LIN {X 0,Y 573.238,Z 498.079,A -85,B 0,C 180,E1 -2309.114,E2 -2309.114} C_VEL
LIN {X 0,Y 573.258,Z 498.071,A -85,B 0,C 180,E1 -2311.967,E2 -2311.967} C_VEL
LIN {X 0,Y 573.252,Z 498.078,A -85,B 0,C 180,E1 -2314.589,E2 -2314.589} C_VEL
LIN {X 0,Y 573.231,Z 498.075,A -85,B 0,C 180,E1 -2317.662,E2 -2317.662} C_VEL
LIN {X 0,Y 573.249,Z 498.072,A -85,B 0,C 180,E1 -2319.923,E2 -2319.923} C_VEL
LIN {X 0,Y 573.254,Z 498.081,A -85,B 0,C 180,E1 -2322.988,E2 -2322.988} C_VEL
LIN {X 0,Y 573.263,Z 498.071,A -85,B 0,C 180,E1 -2325.806,E2 -2325.806} C_VEL
LIN {X 0,Y 573.274,Z 498.076,A -85,B 0,C 180,E1 -2328.734,E2 -2328.734} C_VEL
LIN {X 0,Y 573.299,Z 498.068,A -85,B 0,C 180,E1 -2331.54,E2 -2331.54} C_VEL
LIN {X 0,Y 573.291,Z 498.068,A -85,B 0,C 180,E1 -2334.371,E2 -2334.371} C_VEL
LIN {X 0,Y 573.3,Z 498.066,A -85,B 0,C 180,E1 -2337.892,E2 -2337.892} C_VEL
LIN {X 0,Y 573.329,Z 498.067,A -85,B 0,C 180,E1 -2340.702,E2 -2340.702} C_VEL
LIN {X 0,Y 573.239,Z 498.077,A -85,B 0,C 180,E1 -2343.514,E2 -2343.514} C_VEL
LIN {X 0,Y 573.294,Z 498.069,A -85,B 0,C 180,E1 -2345.628,E2 -2345.628} C_VEL
LIN {X 0,Y 573.299,Z 498.068,A -85,B 0,C 180,E1 -2348.459,E2 -2348.459} C_VEL
LIN {X 0,Y 573.288,Z 498.074,A -85,B 0,C 180,E1 -2351.311,E2 -2351.311} C_VEL
LIN {X 0,Y 573.27,Z 498.071,A -85,B 0,C 180,E1 -2354.425,E2 -2354.425} C_VEL
LIN {X 0,Y 573.25,Z 498.083,A -85,B 0,C 180,E1 -2357.111,E2 -2357.111} C_VEL
LIN {X 0,Y 573.248,Z 498.073,A -85,B 0,C 180,E1 -2360.076,E2 -2360.076} C_VEL
LIN {X 0,Y 573.23,Z 498.076,A -85,B 0,C 180,E1 -2362.338,E2 -2362.338} C_VEL
LIN {X 0,Y 573.242,Z 498.075,A -85,B 0,C 180,E1 -2364.401,E2 -2364.401} C_VEL
LIN {X 0,Y 572.616,Z 498.16,A -85,B 0,C 180,E1 -2364.988,E2 -2364.988} C_VEL
LIN {X 0,Y 569.779,Z 498.518,A -85,B 0,C 180,E1 -2365.939,E2 -2365.939} C_VEL
LIN {X 0,Y 567.351,Z 498.821,A -85,B 0,C 180,E1 -2366.705,E2 -2366.705} C_VEL
LIN {X 0,Y 566.298,Z 498.949,A -85,B 0,C 180,E1 -2367.297,E2 -2367.297} C_VEL
LIN {X 0,Y 566.208,Z 498.956,A -85,B 0,C 180,E1 -2367.497,E2 -2367.497} C_VEL
LIN {X 0,Y 566.186,Z 498.955,A -85,B 0,C 180,E1 -2370.592,E2 -2370.592} C_VEL
LIN {X 0,Y 566.22,Z 498.958,A -85,B 0,C 180,E1 -2373.102,E2 -2373.102} C_VEL
LIN {X 0,Y 566.261,Z 499.123,A -85,B 0,C 180,E1 -2374.382,E2 -2374.382} C_VEL
LIN {X 0,Y 566.267,Z 510.219,A -85,B 0,C 180,E1 -2376.564,E2 -2376.564} C_VEL
LIN {X 0,Y 566.196,Z 517.853,A -85,B 0,C 180,E1 -2378.051,E2 -2378.051} C_VEL
LIN {X 0,Y 567.197,Z 524.442,A -85,B 0,C 180,E1 -2378.169,E2 -2378.169} C_VEL
LIN {X 0,Y 566.927,Z 624.641,A -85,B 0,C 180,E1 -2379.461,E2 -2379.461} C_VEL
LIN {X 0,Y 566.843,Z 638.116,A -85,B 0,C 180,E1 -2379.791,E2 -2379.791} C_VEL
LIN {X 0,Y 566.739,Z 649.818,A -85,B 0,C 180,E1 -2380.211,E2 -2380.211} C_VEL
LIN {X 0,Y 566.583,Z 661.36,A -85,B 0,C 180,E1 -2380.764,E2 -2380.764} C_VEL
LIN {X 0,Y 566.456,Z 672.754,A -85,B 0,C 180,E1 -2381.469,E2 -2381.469} C_VEL
LIN {X 0,Y 566.307,Z 683.695,A -85,B 0,C 180,E1 -2382.318,E2 -2382.318} C_VEL
LIN {X 0,Y 566.189,Z 693.549,A -85,B 0,C 180,E1 -2383.273,E2 -2383.273} C_VEL
LIN {X 0,Y 566.069,Z 701.912,A -85,B 0,C 180,E1 -2384.272,E2 -2384.272} C_VEL
LIN {X 0,Y 566.024,Z 708.75,A -85,B 0,C 180,E1 -2385.273,E2 -2385.273} C_VEL
LIN {X 0,Y 565.94,Z 715.445,A -85,B 0,C 180,E1 -2386.498,E2 -2386.498} C_VEL
LIN {X 0,Y 565.918,Z 719.703,A -85,B 0,C 180,E1 -2387.498,E2 -2387.498} C_VEL
LIN {X 0,Y 565.921,Z 722.017,A -85,B 0,C 180,E1 -2388.169,E2 -2388.169} C_VEL
LIN {X 0,Y 565.836,Z 724.94,A -85,B 0,C 180,E1 -2389.257,E2 -2389.257} C_VEL
LIN {X 0,Y 565.848,Z 726.888,A -85,B 0,C 180,E1 -2390.358,E2 -2390.358} C_VEL
LIN {X 0,Y 565.827,Z 727.91,A -85,B 0,C 180,E1 -2391.609,E2 -2391.609} C_VEL
LIN {X 0,Y 565.828,Z 727.856,A -85,B 0,C 180,E1 -2392.648,E2 -2392.648} C_VEL
LIN {X 0,Y 565.816,Z 726.731,A -85,B 0,C 180,E1 -2393.839,E2 -2393.839} C_VEL
LIN {X 0,Y 565.872,Z 724.149,A -85,B 0,C 180,E1 -2395.159,E2 -2395.159} C_VEL
LIN {X 0,Y 565.916,Z 720.706,A -85,B 0,C 180,E1 -2396.31,E2 -2396.31} C_VEL
LIN {X 0,Y 565.946,Z 715.36,A -85,B 0,C 180,E1 -2397.61,E2 -2397.61} C_VEL
LIN {X 0,Y 565.995,Z 708.949,A -85,B 0,C 180,E1 -2398.786,E2 -2398.786} C_VEL
LIN {X 0,Y 566.094,Z 701.93,A -85,B 0,C 180,E1 -2399.815,E2 -2399.815} C_VEL
LIN {X 0,Y 566.175,Z 693.319,A -85,B 0,C 180,E1 -2400.843,E2 -2400.843} C_VEL
LIN {X 0,Y 566.319,Z 683.652,A -85,B 0,C 180,E1 -2401.775,E2 -2401.775} C_VEL
LIN {X 0,Y 566.432,Z 673.445,A -85,B 0,C 180,E1 -2402.573,E2 -2402.573} C_VEL
LIN {X 0,Y 566.569,Z 662.396,A -85,B 0,C 180,E1 -2403.267,E2 -2403.267} C_VEL
LIN {X 0,Y 566.717,Z 650.965,A -85,B 0,C 180,E1 -2403.832,E2 -2403.832} C_VEL
LIN {X 0,Y 566.828,Z 638.084,A -85,B 0,C 180,E1 -2404.301,E2 -2404.301} C_VEL
LIN {X 0,Y 566.939,Z 625.415,A -85,B 0,C 180,E1 -2404.613,E2 -2404.613} C_VEL
LIN {X 0,Y 567.029,Z 594.146,A -85,B 0,C 180,E1 -2405.036,E2 -2405.036} C_VEL
LIN {X 0,Y 567.13,Z 523.477,A -85,B 0,C 180,E1 -2405.935,E2 -2405.935} C_VEL
LIN {X 0,Y 566.222,Z 517.846,A -85,B 0,C 180,E1 -2406.04,E2 -2406.04} C_VEL
LIN {X 0,Y 566.357,Z 503.159,A -85,B 0,C 180,E1 -2408.909,E2 -2408.909} C_VEL
LIN {X 0,Y 566.225,Z 498.953,A -85,B 0,C 180,E1 -2409.759,E2 -2409.759} C_VEL
LIN {X 0,Y 566.222,Z 498.958,A -85,B 0,C 180,E1 -2412.886,E2 -2412.886} C_VEL
LIN {X 0,Y 566.231,Z 498.947,A -85,B 0,C 180,E1 -2415.627,E2 -2415.627} C_VEL
LIN {X 0,Y 566.232,Z 498.953,A -85,B 0,C 180,E1 -2418.675,E2 -2418.675} C_VEL
LIN {X 0,Y 566.226,Z 498.95,A -85,B 0,C 180,E1 -2421.434,E2 -2421.434} C_VEL
LIN {X 0,Y 566.263,Z 498.944,A -85,B 0,C 180,E1 -2424.302,E2 -2424.302} C_VEL
LIN {X 0,Y 566.282,Z 498.94,A -85,B 0,C 180,E1 -2427.866,E2 -2427.866} C_VEL
LIN {X 0,Y 566.302,Z 498.945,A -85,B 0,C 180,E1 -2430.711,E2 -2430.711} C_VEL
LIN {X 0,Y 566.271,Z 498.951,A -85,B 0,C 180,E1 -2432.845,E2 -2432.845} C_VEL
LIN {X 0,Y 566.264,Z 498.943,A -85,B 0,C 180,E1 -2435.698,E2 -2435.698} C_VEL
LIN {X 0,Y 566.231,Z 498.951,A -85,B 0,C 180,E1 -2438.565,E2 -2438.565} C_VEL
LIN {X 0,Y 566.239,Z 498.948,A -85,B 0,C 180,E1 -2441.454,E2 -2441.454} C_VEL
LIN {X 0,Y 566.231,Z 498.95,A -85,B 0,C 180,E1 -2444.507,E2 -2444.507} C_VEL
LIN {X 0,Y 566.2,Z 498.955,A -85,B 0,C 180,E1 -2447.331,E2 -2447.331} C_VEL
LIN {X 0,Y 566.211,Z 498.951,A -85,B 0,C 180,E1 -2450.337,E2 -2450.337} C_VEL
LIN {X 0,Y 566.185,Z 498.956,A -85,B 0,C 180,E1 -2453.403,E2 -2453.403} C_VEL
LIN {X 0,Y 566.21,Z 498.95,A -85,B 0,C 180,E1 -2455.749,E2 -2455.749} C_VEL
LIN {X 0,Y 566.201,Z 498.951,A -85,B 0,C 180,E1 -2458.203,E2 -2458.203} C_VEL
LIN {X 0,Y 566.19,Z 498.955,A -85,B 0,C 180,E1 -2460.591,E2 -2460.591} C_VEL
LIN {X 0,Y 566.223,Z 498.957,A -85,B 0,C 180,E1 -2463.101,E2 -2463.101} C_VEL
LIN {X 0,Y 566.206,Z 498.951,A -85,B 0,C 180,E1 -2465.688,E2 -2465.688} C_VEL
LIN {X 0,Y 566.211,Z 498.952,A -85,B 0,C 180,E1 -2468.559,E2 -2468.559} C_VEL
LIN {X 0,Y 566.214,Z 498.958,A -85,B 0,C 180,E1 -2471.135,E2 -2471.135} C_VEL
LIN {X 0,Y 566.193,Z 498.951,A -85,B 0,C 180,E1 -2474.035,E2 -2474.035} C_VEL
LIN {X 0,Y 566.197,Z 498.961,A -85,B 0,C 180,E1 -2477.082,E2 -2477.082} C_VEL
LIN {X 0,Y 566.219,Z 498.949,A -85,B 0,C 180,E1 -2479.802,E2 -2479.802} C_VEL
LIN {X 0,Y 566.19,Z 498.955,A -85,B 0,C 180,E1 -2482.599,E2 -2482.599} C_VEL
LIN {X 0,Y 566.215,Z 498.958,A -85,B 0,C 180,E1 -2485.183,E2 -2485.183} C_VEL
LIN {X 0,Y 566.226,Z 498.949,A -85,B 0,C 180,E1 -2487.744,E2 -2487.744} C_VEL
LIN {X 0,Y 566.22,Z 498.949,A -85,B 0,C 180,E1 -2490.323,E2 -2490.323} C_VEL
LIN {X 0,Y 566.228,Z 498.954,A -85,B 0,C 180,E1 -2493.334,E2 -2493.334} C_VEL
LIN {X 0,Y 566.19,Z 498.953,A -85,B 0,C 180,E1 -2495.819,E2 -2495.819} C_VEL
LIN {X 0,Y 566.207,Z 498.956,A -85,B 0,C 180,E1 -2498.903,E2 -2498.903} C_VEL
LIN {X 0,Y 566.205,Z 498.96,A -85,B 0,C 180,E1 -2501.173,E2 -2501.173} C_VEL
LIN {X 0,Y 566.212,Z 498.955,A -85,B 0,C 180,E1 -2503.413,E2 -2503.413} C_VEL
LIN {X 0,Y 566.192,Z 498.952,A -85,B 0,C 180,E1 -2506.359,E2 -2506.359} C_VEL
LIN {X 0,Y 566.264,Z 498.945,A -85,B 0,C 180,E1 -2508.654,E2 -2508.654} C_VEL
LIN {X 0,Y 566.241,Z 498.951,A -85,B 0,C 180,E1 -2511.435,E2 -2511.435} C_VEL
LIN {X 0,Y 566.259,Z 498.943,A -85,B 0,C 180,E1 -2514.302,E2 -2514.302} C_VEL
LIN {X 0,Y 566.271,Z 498.943,A -85,B 0,C 180,E1 -2517.867,E2 -2517.867} C_VEL
LIN {X 0,Y 566.3,Z 498.941,A -85,B 0,C 180,E1 -2520.711,E2 -2520.711} C_VEL
LIN {X 0,Y 566.274,Z 498.946,A -85,B 0,C 180,E1 -2522.846,E2 -2522.846} C_VEL
LIN {X 0,Y 566.263,Z 498.946,A -85,B 0,C 180,E1 -2525.699,E2 -2525.699} C_VEL
LIN {X 0,Y 566.242,Z 498.946,A -85,B 0,C 180,E1 -2528.566,E2 -2528.566} C_VEL
LIN {X 0,Y 566.242,Z 498.952,A -85,B 0,C 180,E1 -2531.455,E2 -2531.455} C_VEL
LIN {X 0,Y 566.225,Z 498.948,A -85,B 0,C 180,E1 -2534.508,E2 -2534.508} C_VEL
LIN {X 0,Y 566.198,Z 498.96,A -85,B 0,C 180,E1 -2537.332,E2 -2537.332} C_VEL
LIN {X 0,Y 566.212,Z 498.949,A -85,B 0,C 180,E1 -2540.338,E2 -2540.338} C_VEL
LIN {X 0,Y 566.182,Z 498.961,A -85,B 0,C 180,E1 -2543.405,E2 -2543.405} C_VEL
LIN {X 0,Y 566.219,Z 498.951,A -85,B 0,C 180,E1 -2545.749,E2 -2545.749} C_VEL
LIN {X 0,Y 566.2,Z 498.951,A -85,B 0,C 180,E1 -2548.204,E2 -2548.204} C_VEL
LIN {X 0,Y 566.188,Z 498.953,A -85,B 0,C 180,E1 -2550.593,E2 -2550.593} C_VEL
LIN {X 0,Y 566.223,Z 498.954,A -85,B 0,C 180,E1 -2553.102,E2 -2553.102} C_VEL
LIN {X 0,Y 566.208,Z 498.954,A -85,B 0,C 180,E1 -2555.689,E2 -2555.689} C_VEL
LIN {X 0,Y 566.212,Z 498.95,A -85,B 0,C 180,E1 -2558.56,E2 -2558.56} C_VEL
LIN {X 0,Y 566.208,Z 498.956,A -85,B 0,C 180,E1 -2561.137,E2 -2561.137} C_VEL
LIN {X 0,Y 566.196,Z 498.952,A -85,B 0,C 180,E1 -2564.036,E2 -2564.036} C_VEL
LIN {X 0,Y 566.207,Z 498.955,A -85,B 0,C 180,E1 -2567.083,E2 -2567.083} C_VEL
LIN {X 0,Y 566.225,Z 498.951,A -85,B 0,C 180,E1 -2569.804,E2 -2569.804} C_VEL
LIN {X 0,Y 566.198,Z 498.951,A -85,B 0,C 180,E1 -2572.6,E2 -2572.6} C_VEL
LIN {X 0,Y 566.209,Z 498.956,A -85,B 0,C 180,E1 -2575.183,E2 -2575.183} C_VEL
LIN {X 0,Y 566.234,Z 498.952,A -85,B 0,C 180,E1 -2577.745,E2 -2577.745} C_VEL
LIN {X 0,Y 566.204,Z 498.951,A -85,B 0,C 180,E1 -2580.329,E2 -2580.329} C_VEL
LIN {X 0,Y 566.212,Z 498.952,A -85,B 0,C 180,E1 -2582.662,E2 -2582.662} C_VEL
LIN {X 0,Y 566.249,Z 499.022,A -85,B 0,C 180,E1 -2585.456,E2 -2585.456} C_VEL
LIN {X 0,Y 567.269,Z 504.225,A -85,B 0,C 180,E1 -2586.221,E2 -2586.221} C_VEL
LIN {X 0,Y 567.127,Z 520.193,A -85,B 0,C 180,E1 -2588.465,E2 -2588.465} C_VEL
LIN {X 0,Y 566.837,Z 539.96,A -85,B 0,C 180,E1 -2591.195,E2 -2591.195} C_VEL
LIN {X 0,Y 566.582,Z 560.431,A -85,B 0,C 180,E1 -2593.979,E2 -2593.979} C_VEL
LIN {X 0,Y 566.428,Z 575.357,A -85,B 0,C 180,E1 -2595.987,E2 -2595.987} C_VEL
LIN {X 0,Y 567.197,Z 581.535,A -85,B 0,C 180,E1 -2596.087,E2 -2596.087} C_VEL
LIN {X 0,Y 566.921,Z 683.962,A -85,B 0,C 180,E1 -2597.403,E2 -2597.403} C_VEL
LIN {X 0,Y 566.848,Z 697.229,A -85,B 0,C 180,E1 -2597.719,E2 -2597.719} C_VEL
LIN {X 0,Y 566.758,Z 709.382,A -85,B 0,C 180,E1 -2598.149,E2 -2598.149} C_VEL
LIN {X 0,Y 566.627,Z 721.158,A -85,B 0,C 180,E1 -2598.708,E2 -2598.708} C_VEL
LIN {X 0,Y 566.458,Z 733.205,A -85,B 0,C 180,E1 -2599.456,E2 -2599.456} C_VEL
LIN {X 0,Y 566.318,Z 743.604,A -85,B 0,C 180,E1 -2600.266,E2 -2600.266} C_VEL
LIN {X 0,Y 566.207,Z 752.115,A -85,B 0,C 180,E1 -2601.074,E2 -2601.074} C_VEL
LIN {X 0,Y 566.112,Z 759.962,A -85,B 0,C 180,E1 -2601.972,E2 -2601.972} C_VEL
LIN {X 0,Y 566.004,Z 767.623,A -85,B 0,C 180,E1 -2603.047,E2 -2603.047} C_VEL
LIN {X 0,Y 566.004,Z 774.681,A -85,B 0,C 180,E1 -2604.299,E2 -2604.299} C_VEL
LIN {X 0,Y 565.933,Z 779.372,A -85,B 0,C 180,E1 -2605.37,E2 -2605.37} C_VEL
LIN {X 0,Y 565.927,Z 782.958,A -85,B 0,C 180,E1 -2606.44,E2 -2606.44} C_VEL
LIN {X 0,Y 565.878,Z 784.808,A -85,B 0,C 180,E1 -2607.153,E2 -2607.153} C_VEL
LIN {X 0,Y 565.846,Z 787.186,A -85,B 0,C 180,E1 -2608.577,E2 -2608.577} C_VEL
LIN {X 0,Y 565.839,Z 788,A -85,B 0,C 180,E1 -2610,E2 -2610} C_VEL
LIN {X 0,Y 565.846,Z 787.186,A -85,B 0,C 180,E1 -2611.423,E2 -2611.423} C_VEL
LIN {X 0,Y 565.878,Z 784.81,A -85,B 0,C 180,E1 -2612.847,E2 -2612.847} C_VEL
LIN {X 0,Y 565.926,Z 781.896,A -85,B 0,C 180,E1 -2613.916,E2 -2613.916} C_VEL
LIN {X 0,Y 565.878,Z 777.949,A -85,B 0,C 180,E1 -2614.987,E2 -2614.987} C_VEL
LIN {X 0,Y 566.002,Z 772.867,A -85,B 0,C 180,E1 -2616.058,E2 -2616.058} C_VEL
LIN {X 0,Y 566.04,Z 766.47,A -85,B 0,C 180,E1 -2617.132,E2 -2617.132} C_VEL
LIN {X 0,Y 566.134,Z 758.48,A -85,B 0,C 180,E1 -2618.207,E2 -2618.207} C_VEL
LIN {X 0,Y 566.228,Z 750.338,A -85,B 0,C 180,E1 -2619.105,E2 -2619.105} C_VEL
LIN {X 0,Y 566.341,Z 740.404,A -85,B 0,C 180,E1 -2620.005,E2 -2620.005} C_VEL
LIN {X 0,Y 566.523,Z 729.288,A -85,B 0,C 180,E1 -2620.807,E2 -2620.807} C_VEL
LIN {X 0,Y 566.66,Z 718.182,A -85,B 0,C 180,E1 -2621.445,E2 -2621.445} C_VEL
LIN {X 0,Y 566.735,Z 705.991,A -85,B 0,C 180,E1 -2621.988,E2 -2621.988} C_VEL
LIN {X 0,Y 566.879,Z 693.188,A -85,B 0,C 180,E1 -2622.394,E2 -2622.394} C_VEL
LIN {X 0,Y 566.988,Z 681.127,A -85,B 0,C 180,E1 -2622.641,E2 -2622.641} C_VEL
LIN {X 0,Y 567.056,Z 579.746,A -85,B 0,C 180,E1 -2623.94,E2 -2623.94} C_VEL
LIN {X 0,Y 566.446,Z 575.272,A -85,B 0,C 180,E1 -2624.024,E2 -2624.024} C_VEL
LIN {X 0,Y 566.673,Z 552.206,A -85,B 0,C 180,E1 -2627.135,E2 -2627.135} C_VEL
LIN {X 0,Y 566.955,Z 530.408,A -85,B 0,C 180,E1 -2630.119,E2 -2630.119} C_VEL
LIN {X 0,Y 567.305,Z 509.936,A -85,B 0,C 180,E1 -2632.969,E2 -2632.969} C_VEL
LIN {X 0,Y 567.276,Z 504.204,A -85,B 0,C 180,E1 -2633.782,E2 -2633.782} C_VEL
LIN {X 0,Y 566.257,Z 498.954,A -85,B 0,C 180,E1 -2634.568,E2 -2634.568} C_VEL
LIN {X 0,Y 566.212,Z 498.952,A -85,B 0,C 180,E1 -2637.338,E2 -2637.338} C_VEL
LIN {X 0,Y 566.202,Z 498.952,A -85,B 0,C 180,E1 -2639.768,E2 -2639.768} C_VEL
LIN {X 0,Y 566.207,Z 498.958,A -85,B 0,C 180,E1 -2642.43,E2 -2642.43} C_VEL
LIN {X 0,Y 566.212,Z 498.955,A -85,B 0,C 180,E1 -2644.994,E2 -2644.994} C_VEL
LIN {X 0,Y 566.196,Z 498.952,A -85,B 0,C 180,E1 -2647.46,E2 -2647.46} C_VEL
LIN {X 0,Y 566.225,Z 498.951,A -85,B 0,C 180,E1 -2650.196,E2 -2650.196} C_VEL
LIN {X 0,Y 566.207,Z 498.955,A -85,B 0,C 180,E1 -2653.052,E2 -2653.052} C_VEL
LIN {X 0,Y 566.198,Z 498.952,A -85,B 0,C 180,E1 -2656.047,E2 -2656.047} C_VEL
LIN {X 0,Y 566.207,Z 498.958,A -85,B 0,C 180,E1 -2658.863,E2 -2658.863} C_VEL
LIN {X 0,Y 566.186,Z 498.953,A -85,B 0,C 180,E1 -2661.636,E2 -2661.636} C_VEL
LIN {X 0,Y 566.208,Z 498.953,A -85,B 0,C 180,E1 -2664.311,E2 -2664.311} C_VEL
LIN {X 0,Y 566.223,Z 498.957,A -85,B 0,C 180,E1 -2666.898,E2 -2666.898} C_VEL
LIN {X 0,Y 566.188,Z 498.954,A -85,B 0,C 180,E1 -2669.407,E2 -2669.407} C_VEL
LIN {X 0,Y 566.221,Z 498.948,A -85,B 0,C 180,E1 -2671.858,E2 -2671.858} C_VEL
LIN {X 0,Y 566.22,Z 498.95,A -85,B 0,C 180,E1 -2674.251,E2 -2674.251} C_VEL
LIN {X 0,Y 566.185,Z 498.959,A -85,B 0,C 180,E1 -2676.713,E2 -2676.713} C_VEL
LIN {X 0,Y 566.212,Z 498.949,A -85,B 0,C 180,E1 -2679.662,E2 -2679.662} C_VEL
LIN {X 0,Y 566.196,Z 498.957,A -85,B 0,C 180,E1 -2682.668,E2 -2682.668} C_VEL
LIN {X 0,Y 566.224,Z 498.948,A -85,B 0,C 180,E1 -2685.626,E2 -2685.626} C_VEL
LIN {X 0,Y 566.266,Z 498.948,A -85,B 0,C 180,E1 -2688.653,E2 -2688.653} C_VEL
LIN {X 0,Y 566.24,Z 498.949,A -85,B 0,C 180,E1 -2691.434,E2 -2691.434} C_VEL
LIN {X 0,Y 566.259,Z 498.944,A -85,B 0,C 180,E1 -2694.301,E2 -2694.301} C_VEL
LIN {X 0,Y 566.271,Z 498.942,A -85,B 0,C 180,E1 -2697.866,E2 -2697.866} C_VEL
LIN {X 0,Y 566.299,Z 498.943,A -85,B 0,C 180,E1 -2700.711,E2 -2700.711} C_VEL
LIN {X 0,Y 566.272,Z 498.949,A -85,B 0,C 180,E1 -2702.845,E2 -2702.845} C_VEL
LIN {X 0,Y 566.262,Z 498.944,A -85,B 0,C 180,E1 -2705.698,E2 -2705.698} C_VEL
LIN {X 0,Y 566.241,Z 498.948,A -85,B 0,C 180,E1 -2708.565,E2 -2708.565} C_VEL
LIN {X 0,Y 566.24,Z 498.95,A -85,B 0,C 180,E1 -2711.454,E2 -2711.454} C_VEL
LIN {X 0,Y 566.223,Z 498.95,A -85,B 0,C 180,E1 -2714.507,E2 -2714.507} C_VEL
LIN {X 0,Y 566.195,Z 498.959,A -85,B 0,C 180,E1 -2717.331,E2 -2717.331} C_VEL
LIN {X 0,Y 566.211,Z 498.95,A -85,B 0,C 180,E1 -2720.337,E2 -2720.337} C_VEL
LIN {X 0,Y 566.18,Z 498.961,A -85,B 0,C 180,E1 -2723.404,E2 -2723.404} C_VEL
LIN {X 0,Y 566.218,Z 498.952,A -85,B 0,C 180,E1 -2725.748,E2 -2725.748} C_VEL
LIN {X 0,Y 566.208,Z 498.956,A -85,B 0,C 180,E1 -2727.497,E2 -2727.497} C_VEL
LIN {X 0,Y 565.529,Z 499.038,A -85,B 0,C 180,E1 -2728.091,E2 -2728.091} C_VEL
LIN {X 0,Y 562.664,Z 499.401,A -85,B 0,C 180,E1 -2729.054,E2 -2729.054} C_VEL
LIN {X 0,Y 560.253,Z 499.696,A -85,B 0,C 180,E1 -2729.83,E2 -2729.83} C_VEL
LIN {X 0,Y 559.225,Z 499.822,A -85,B 0,C 180,E1 -2730.429,E2 -2730.429} C_VEL
LIN {X 0,Y 559.144,Z 499.833,A -85,B 0,C 180,E1 -2730.631,E2 -2730.631} C_VEL
LIN {X 0,Y 559.168,Z 499.835,A -85,B 0,C 180,E1 -2733.574,E2 -2733.574} C_VEL
LIN {X 0,Y 559.223,Z 499.985,A -85,B 0,C 180,E1 -2734.325,E2 -2734.325} C_VEL
LIN {X 0,Y 559.247,Z 510.703,A -85,B 0,C 180,E1 -2736.461,E2 -2736.461} C_VEL
LIN {X 0,Y 559.188,Z 517.827,A -85,B 0,C 180,E1 -2737.867,E2 -2737.867} C_VEL
LIN {X 0,Y 560.336,Z 525.282,A -85,B 0,C 180,E1 -2738.006,E2 -2738.006} C_VEL
LIN {X 0,Y 560.038,Z 624.109,A -85,B 0,C 180,E1 -2739.293,E2 -2739.293} C_VEL
LIN {X 0,Y 559.894,Z 637.137,A -85,B 0,C 180,E1 -2739.607,E2 -2739.607} C_VEL
LIN {X 0,Y 559.783,Z 650.179,A -85,B 0,C 180,E1 -2740.077,E2 -2740.077} C_VEL
LIN {X 0,Y 559.589,Z 662.251,A -85,B 0,C 180,E1 -2740.672,E2 -2740.672} C_VEL
LIN {X 0,Y 559.443,Z 673.522,A -85,B 0,C 180,E1 -2741.389,E2 -2741.389} C_VEL
LIN {X 0,Y 559.273,Z 684.342,A -85,B 0,C 180,E1 -2742.251,E2 -2742.251} C_VEL
LIN {X 0,Y 559.137,Z 693.869,A -85,B 0,C 180,E1 -2743.197,E2 -2743.197} C_VEL
LIN {X 0,Y 559.006,Z 702.977,A -85,B 0,C 180,E1 -2744.316,E2 -2744.316} C_VEL
LIN {X 0,Y 558.94,Z 709.091,A -85,B 0,C 180,E1 -2745.242,E2 -2745.242} C_VEL
LIN {X 0,Y 558.874,Z 714.53,A -85,B 0,C 180,E1 -2746.241,E2 -2746.241} C_VEL
LIN {X 0,Y 558.839,Z 718.865,A -85,B 0,C 180,E1 -2747.227,E2 -2747.227} C_VEL
LIN {X 0,Y 558.819,Z 722.252,A -85,B 0,C 180,E1 -2748.199,E2 -2748.199} C_VEL
LIN {X 0,Y 558.756,Z 724.792,A -85,B 0,C 180,E1 -2749.153,E2 -2749.153} C_VEL
LIN {X 0,Y 558.756,Z 726.547,A -85,B 0,C 180,E1 -2750.107,E2 -2750.107} C_VEL
LIN {X 0,Y 558.725,Z 727.737,A -85,B 0,C 180,E1 -2751.248,E2 -2751.248} C_VEL
LIN {X 0,Y 558.735,Z 727.926,A -85,B 0,C 180,E1 -2752.413,E2 -2752.413} C_VEL
LIN {X 0,Y 558.719,Z 726.879,A -85,B 0,C 180,E1 -2753.759,E2 -2753.759} C_VEL
LIN {X 0,Y 558.762,Z 724.994,A -85,B 0,C 180,E1 -2754.84,E2 -2754.84} C_VEL
LIN {X 0,Y 558.813,Z 721.597,A -85,B 0,C 180,E1 -2756.104,E2 -2756.104} C_VEL
LIN {X 0,Y 558.856,Z 716.567,A -85,B 0,C 180,E1 -2757.412,E2 -2757.412} C_VEL
LIN {X 0,Y 558.919,Z 711.258,A -85,B 0,C 180,E1 -2758.473,E2 -2758.473} C_VEL
LIN {X 0,Y 558.989,Z 704.215,A -85,B 0,C 180,E1 -2759.6,E2 -2759.6} C_VEL
LIN {X 0,Y 559.109,Z 696.087,A -85,B 0,C 180,E1 -2760.645,E2 -2760.645} C_VEL
LIN {X 0,Y 559.234,Z 686.864,A -85,B 0,C 180,E1 -2761.606,E2 -2761.606} C_VEL
LIN {X 0,Y 559.42,Z 676.213,A -85,B 0,C 180,E1 -2762.505,E2 -2762.505} C_VEL
LIN {X 0,Y 559.556,Z 665.137,A -85,B 0,C 180,E1 -2763.25,E2 -2763.25} C_VEL
LIN {X 0,Y 559.712,Z 653.158,A -85,B 0,C 180,E1 -2763.88,E2 -2763.88} C_VEL
LIN {X 0,Y 559.893,Z 640.397,A -85,B 0,C 180,E1 -2764.383,E2 -2764.383} C_VEL
LIN {X 0,Y 560.011,Z 628.043,A -85,B 0,C 180,E1 -2764.718,E2 -2764.718} C_VEL
LIN {X 0,Y 560.089,Z 611.02,A -85,B 0,C 180,E1 -2764.982,E2 -2764.982} C_VEL
LIN {X 0,Y 560.287,Z 524.896,A -85,B 0,C 180,E1 -2766.09,E2 -2766.09} C_VEL
LIN {X 0,Y 559.177,Z 517.889,A -85,B 0,C 180,E1 -2766.212,E2 -2766.212} C_VEL
LIN {X 0,Y 559.324,Z 503.713,A -85,B 0,C 180,E1 -2769.017,E2 -2769.017} C_VEL
LIN {X 0,Y 559.201,Z 499.829,A -85,B 0,C 180,E1 -2769.829,E2 -2769.829} C_VEL
LIN {X 0,Y 559.179,Z 499.831,A -85,B 0,C 180,E1 -2773.198,E2 -2773.198} C_VEL
LIN {X 0,Y 559.171,Z 499.827,A -85,B 0,C 180,E1 -2776.184,E2 -2776.184} C_VEL
LIN {X 0,Y 559.192,Z 499.83,A -85,B 0,C 180,E1 -2779.134,E2 -2779.134} C_VEL
LIN {X 0,Y 559.204,Z 499.822,A -85,B 0,C 180,E1 -2782.054,E2 -2782.054} C_VEL
LIN {X 0,Y 559.252,Z 499.826,A -85,B 0,C 180,E1 -2784.953,E2 -2784.953} C_VEL
LIN {X 0,Y 559.253,Z 499.816,A -85,B 0,C 180,E1 -2787.839,E2 -2787.839} C_VEL
LIN {X 0,Y 559.272,Z 499.82,A -85,B 0,C 180,E1 -2790.72,E2 -2790.72} C_VEL
LIN {X 0,Y 559.237,Z 499.828,A -85,B 0,C 180,E1 -2792.881,E2 -2792.881} C_VEL
LIN {X 0,Y 559.234,Z 499.819,A -85,B 0,C 180,E1 -2795.77,E2 -2795.77} C_VEL
LIN {X 0,Y 559.189,Z 499.83,A -85,B 0,C 180,E1 -2798.674,E2 -2798.674} C_VEL
LIN {X 0,Y 559.203,Z 499.824,A -85,B 0,C 180,E1 -2801.6,E2 -2801.6} C_VEL
LIN {X 0,Y 559.197,Z 499.827,A -85,B 0,C 180,E1 -2804.595,E2 -2804.595} C_VEL
LIN {X 0,Y 559.16,Z 499.829,A -85,B 0,C 180,E1 -2807.556,E2 -2807.556} C_VEL
LIN {X 0,Y 559.169,Z 499.827,A -85,B 0,C 180,E1 -2809.837,E2 -2809.837} C_VEL
LIN {X 0,Y 559.138,Z 499.831,A -85,B 0,C 180,E1 -2812.152,E2 -2812.152} C_VEL
LIN {X 0,Y 559.174,Z 499.833,A -85,B 0,C 180,E1 -2815.187,E2 -2815.187} C_VEL
LIN {X 0,Y 559.188,Z 499.825,A -85,B 0,C 180,E1 -2817.711,E2 -2817.711} C_VEL
LIN {X 0,Y 559.164,Z 499.827,A -85,B 0,C 180,E1 -2820.181,E2 -2820.181} C_VEL
LIN {X 0,Y 559.17,Z 499.831,A -85,B 0,C 180,E1 -2822.713,E2 -2822.713} C_VEL
LIN {X 0,Y 559.151,Z 499.834,A -85,B 0,C 180,E1 -2825.321,E2 -2825.321} C_VEL
LIN {X 0,Y 559.13,Z 499.831,A -85,B 0,C 180,E1 -2828.017,E2 -2828.017} C_VEL
LIN {X 0,Y 559.173,Z 499.832,A -85,B 0,C 180,E1 -2830.81,E2 -2830.81} C_VEL
LIN {X 0,Y 559.157,Z 499.829,A -85,B 0,C 180,E1 -2833.731,E2 -2833.731} C_VEL
LIN {X 0,Y 559.16,Z 499.833,A -85,B 0,C 180,E1 -2836.801,E2 -2836.801} C_VEL
LIN {X 0,Y 559.168,Z 499.835,A -85,B 0,C 180,E1 -2839.189,E2 -2839.189} C_VEL
LIN {X 0,Y 559.127,Z 499.832,A -85,B 0,C 180,E1 -2841.982,E2 -2841.982} C_VEL
LIN {X 0,Y 559.151,Z 499.832,A -85,B 0,C 180,E1 -2844.678,E2 -2844.678} C_VEL
LIN {X 0,Y 559.165,Z 499.833,A -85,B 0,C 180,E1 -2847.361,E2 -2847.361} C_VEL
LIN {X 0,Y 559.18,Z 499.825,A -85,B 0,C 180,E1 -2850.135,E2 -2850.135} C_VEL
LIN {X 0,Y 559.174,Z 499.835,A -85,B 0,C 180,E1 -2853.169,E2 -2853.169} C_VEL
LIN {X 0,Y 559.147,Z 499.833,A -85,B 0,C 180,E1 -2855.495,E2 -2855.495} C_VEL
LIN {X 0,Y 559.167,Z 499.829,A -85,B 0,C 180,E1 -2858.624,E2 -2858.624} C_VEL
LIN {X 0,Y 559.162,Z 499.834,A -85,B 0,C 180,E1 -2860.926,E2 -2860.926} C_VEL
LIN {X 0,Y 559.162,Z 499.828,A -85,B 0,C 180,E1 -2863.948,E2 -2863.948} C_VEL
LIN {X 0,Y 559.165,Z 499.827,A -85,B 0,C 180,E1 -2866.184,E2 -2866.184} C_VEL
LIN {X 0,Y 559.223,Z 499.83,A -85,B 0,C 180,E1 -2869.134,E2 -2869.134} C_VEL
LIN {X 0,Y 559.204,Z 499.822,A -85,B 0,C 180,E1 -2872.054,E2 -2872.054} C_VEL
LIN {X 0,Y 559.255,Z 499.822,A -85,B 0,C 180,E1 -2874.954,E2 -2874.954} C_VEL
LIN {X 0,Y 559.243,Z 499.819,A -85,B 0,C 180,E1 -2877.84,E2 -2877.84} C_VEL
LIN {X 0,Y 559.269,Z 499.817,A -85,B 0,C 180,E1 -2880.72,E2 -2880.72} C_VEL
LIN {X 0,Y 559.239,Z 499.822,A -85,B 0,C 180,E1 -2882.882,E2 -2882.882} C_VEL
LIN {X 0,Y 559.232,Z 499.821,A -85,B 0,C 180,E1 -2885.77,E2 -2885.77} C_VEL
LIN {X 0,Y 559.197,Z 499.825,A -85,B 0,C 180,E1 -2888.675,E2 -2888.675} C_VEL
LIN {X 0,Y 559.2,Z 499.827,A -85,B 0,C 180,E1 -2891.601,E2 -2891.601} C_VEL
LIN {X 0,Y 559.19,Z 499.825,A -85,B 0,C 180,E1 -2894.596,E2 -2894.596} C_VEL
LIN {X 0,Y 559.157,Z 499.833,A -85,B 0,C 180,E1 -2897.557,E2 -2897.557} C_VEL
LIN {X 0,Y 559.167,Z 499.829,A -85,B 0,C 180,E1 -2899.838,E2 -2899.838} C_VEL
LIN {X 0,Y 559.135,Z 499.831,A -85,B 0,C 180,E1 -2902.153,E2 -2902.153} C_VEL
LIN {X 0,Y 559.172,Z 499.835,A -85,B 0,C 180,E1 -2905.188,E2 -2905.188} C_VEL
LIN {X 0,Y 559.189,Z 499.828,A -85,B 0,C 180,E1 -2907.712,E2 -2907.712} C_VEL
LIN {X 0,Y 559.163,Z 499.827,A -85,B 0,C 180,E1 -2910.183,E2 -2910.183} C_VEL
LIN {X 0,Y 559.17,Z 499.828,A -85,B 0,C 180,E1 -2912.715,E2 -2912.715} C_VEL
LIN {X 0,Y 559.155,Z 499.839,A -85,B 0,C 180,E1 -2915.322,E2 -2915.322} C_VEL
LIN {X 0,Y 559.13,Z 499.832,A -85,B 0,C 180,E1 -2918.018,E2 -2918.018} C_VEL
LIN {X 0,Y 559.172,Z 499.828,A -85,B 0,C 180,E1 -2920.811,E2 -2920.811} C_VEL
LIN {X 0,Y 559.159,Z 499.832,A -85,B 0,C 180,E1 -2923.733,E2 -2923.733} C_VEL
LIN {X 0,Y 559.168,Z 499.829,A -85,B 0,C 180,E1 -2926.802,E2 -2926.802} C_VEL
LIN {X 0,Y 559.174,Z 499.833,A -85,B 0,C 180,E1 -2929.19,E2 -2929.19} C_VEL
LIN {X 0,Y 559.134,Z 499.832,A -85,B 0,C 180,E1 -2931.984,E2 -2931.984} C_VEL
LIN {X 0,Y 559.146,Z 499.831,A -85,B 0,C 180,E1 -2934.786,E2 -2934.786} C_VEL
LIN {X 0,Y 559.174,Z 499.836,A -85,B 0,C 180,E1 -2937.362,E2 -2937.362} C_VEL
LIN {X 0,Y 559.15,Z 499.831,A -85,B 0,C 180,E1 -2940.143,E2 -2940.143} C_VEL
LIN {X 0,Y 559.17,Z 499.833,A -85,B 0,C 180,E1 -2943.098,E2 -2943.098} C_VEL
LIN {X 0,Y 559.222,Z 499.921,A -85,B 0,C 180,E1 -2945.302,E2 -2945.302} C_VEL
LIN {X 0,Y 560.407,Z 506.958,A -85,B 0,C 180,E1 -2946.341,E2 -2946.341} C_VEL
LIN {X 0,Y 560.127,Z 524.948,A -85,B 0,C 180,E1 -2948.855,E2 -2948.855} C_VEL
LIN {X 0,Y 559.841,Z 544.054,A -85,B 0,C 180,E1 -2951.52,E2 -2951.52} C_VEL
LIN {X 0,Y 559.494,Z 565.89,A -85,B 0,C 180,E1 -2954.519,E2 -2954.519} C_VEL
LIN {X 0,Y 559.439,Z 575.357,A -85,B 0,C 180,E1 -2955.809,E2 -2955.809} C_VEL
LIN {X 0,Y 560.316,Z 582.205,A -85,B 0,C 180,E1 -2955.921,E2 -2955.921} C_VEL
LIN {X 0,Y 560.005,Z 683.962,A -85,B 0,C 180,E1 -2957.244,E2 -2957.244} C_VEL
LIN {X 0,Y 559.927,Z 697.228,A -85,B 0,C 180,E1 -2957.565,E2 -2957.565} C_VEL
LIN {X 0,Y 559.807,Z 709.383,A -85,B 0,C 180,E1 -2957.999,E2 -2957.999} C_VEL
LIN {X 0,Y 559.669,Z 720.815,A -85,B 0,C 180,E1 -2958.547,E2 -2958.547} C_VEL
LIN {X 0,Y 559.495,Z 731.912,A -85,B 0,C 180,E1 -2959.231,E2 -2959.231} C_VEL
LIN {X 0,Y 559.309,Z 742.543,A -85,B 0,C 180,E1 -2960.051,E2 -2960.051} C_VEL
LIN {X 0,Y 559.161,Z 752.115,A -85,B 0,C 180,E1 -2960.961,E2 -2960.961} C_VEL
LIN {X 0,Y 559.05,Z 759.962,A -85,B 0,C 180,E1 -2961.87,E2 -2961.87} C_VEL
LIN {X 0,Y 558.944,Z 767.623,A -85,B 0,C 180,E1 -2962.959,E2 -2962.959} C_VEL
LIN {X 0,Y 558.935,Z 774.68,A -85,B 0,C 180,E1 -2964.227,E2 -2964.227} C_VEL
LIN {X 0,Y 558.827,Z 779.373,A -85,B 0,C 180,E1 -2965.311,E2 -2965.311} C_VEL
LIN {X 0,Y 558.836,Z 782.958,A -85,B 0,C 180,E1 -2966.395,E2 -2966.395} C_VEL
LIN {X 0,Y 558.799,Z 784.808,A -85,B 0,C 180,E1 -2967.116,E2 -2967.116} C_VEL
LIN {X 0,Y 558.745,Z 787.185,A -85,B 0,C 180,E1 -2968.559,E2 -2968.559} C_VEL
LIN {X 0,Y 558.74,Z 788,A -85,B 0,C 180,E1 -2970,E2 -2970} C_VEL
LIN {X 0,Y 558.745,Z 787.186,A -85,B 0,C 180,E1 -2971.441,E2 -2971.441} C_VEL
LIN {X 0,Y 558.799,Z 784.81,A -85,B 0,C 180,E1 -2972.884,E2 -2972.884} C_VEL
LIN {X 0,Y 558.844,Z 781.896,A -85,B 0,C 180,E1 -2973.966,E2 -2973.966} C_VEL
LIN {X 0,Y 558.799,Z 777.949,A -85,B 0,C 180,E1 -2975.051,E2 -2975.051} C_VEL
LIN {X 0,Y 558.921,Z 772.868,A -85,B 0,C 180,E1 -2976.135,E2 -2976.135} C_VEL
LIN {X 0,Y 558.977,Z 766.469,A -85,B 0,C 180,E1 -2977.223,E2 -2977.223} C_VEL
LIN {X 0,Y 559.099,Z 758.48,A -85,B 0,C 180,E1 -2978.311,E2 -2978.311} C_VEL
LIN {X 0,Y 559.184,Z 750.337,A -85,B 0,C 180,E1 -2979.221,E2 -2979.221} C_VEL
LIN {X 0,Y 559.352,Z 740.403,A -85,B 0,C 180,E1 -2980.131,E2 -2980.131} C_VEL
LIN {X 0,Y 559.544,Z 729.368,A -85,B 0,C 180,E1 -2980.939,E2 -2980.939} C_VEL
LIN {X 0,Y 559.703,Z 717.148,A -85,B 0,C 180,E1 -2981.643,E2 -2981.643} C_VEL
LIN {X 0,Y 559.824,Z 704.776,A -85,B 0,C 180,E1 -2982.184,E2 -2982.184} C_VEL
LIN {X 0,Y 559.97,Z 691.359,A -85,B 0,C 180,E1 -2982.595,E2 -2982.595} C_VEL
LIN {X 0,Y 560.086,Z 679.622,A -85,B 0,C 180,E1 -2982.823,E2 -2982.823} C_VEL
LIN {X 0,Y 560.254,Z 581.087,A -85,B 0,C 180,E1 -2984.095,E2 -2984.095} C_VEL
LIN {X 0,Y 559.459,Z 575.272,A -85,B 0,C 180,E1 -2984.202,E2 -2984.202} C_VEL
LIN {X 0,Y 559.708,Z 551.967,A -85,B 0,C 180,E1 -2987.388,E2 -2987.388} C_VEL
LIN {X 0,Y 560.074,Z 530.407,A -85,B 0,C 180,E1 -2990.378,E2 -2990.378} C_VEL
LIN {X 0,Y 560.421,Z 509.731,A -85,B 0,C 180,E1 -2993.267,E2 -2993.267} C_VEL
LIN {X 0,Y 560.075,Z 504.087,A -85,B 0,C 180,E1 -2994.067,E2 -2994.067} C_VEL
LIN {X 0,Y 559.209,Z 499.832,A -85,B 0,C 180,E1 -2994.723,E2 -2994.723} C_VEL
LIN {X 0,Y 559.182,Z 499.827,A -85,B 0,C 180,E1 -2997.711,E2 -2997.711} C_VEL
LIN {X 0,Y 559.157,Z 499.833,A -85,B 0,C 180,E1 -3000.182,E2 -3000.182} C_VEL
LIN {X 0,Y 559.175,Z 499.836,A -85,B 0,C 180,E1 -3002.713,E2 -3002.713} C_VEL
LIN {X 0,Y 559.157,Z 499.831,A -85,B 0,C 180,E1 -3005.321,E2 -3005.321} C_VEL
LIN {X 0,Y 559.134,Z 499.833,A -85,B 0,C 180,E1 -3008.016,E2 -3008.016} C_VEL
LIN {X 0,Y 559.174,Z 499.835,A -85,B 0,C 180,E1 -3010.81,E2 -3010.81} C_VEL
LIN {X 0,Y 559.161,Z 499.828,A -85,B 0,C 180,E1 -3013.731,E2 -3013.731} C_VEL
LIN {X 0,Y 559.164,Z 499.836,A -85,B 0,C 180,E1 -3016.8,E2 -3016.8} C_VEL
LIN {X 0,Y 559.172,Z 499.83,A -85,B 0,C 180,E1 -3019.189,E2 -3019.189} C_VEL
LIN {X 0,Y 559.13,Z 499.832,A -85,B 0,C 180,E1 -3021.982,E2 -3021.982} C_VEL
LIN {X 0,Y 559.156,Z 499.838,A -85,B 0,C 180,E1 -3024.782,E2 -3024.782} C_VEL
LIN {X 0,Y 559.168,Z 499.829,A -85,B 0,C 180,E1 -3027.36,E2 -3027.36} C_VEL
LIN {X 0,Y 559.183,Z 499.826,A -85,B 0,C 180,E1 -3030.134,E2 -3030.134} C_VEL
LIN {X 0,Y 559.177,Z 499.831,A -85,B 0,C 180,E1 -3033.169,E2 -3033.169} C_VEL
LIN {X 0,Y 559.149,Z 499.829,A -85,B 0,C 180,E1 -3035.494,E2 -3035.494} C_VEL
LIN {X 0,Y 559.169,Z 499.833,A -85,B 0,C 180,E1 -3038.623,E2 -3038.623} C_VEL
LIN {X 0,Y 559.18,Z 499.835,A -85,B 0,C 180,E1 -3040.926,E2 -3040.926} C_VEL
LIN {X 0,Y 559.164,Z 499.827,A -85,B 0,C 180,E1 -3043.947,E2 -3043.947} C_VEL
LIN {X 0,Y 559.165,Z 499.827,A -85,B 0,C 180,E1 -3046.184,E2 -3046.184} C_VEL
LIN {X 0,Y 559.203,Z 499.829,A -85,B 0,C 180,E1 -3049.133,E2 -3049.133} C_VEL
LIN {X 0,Y 559.205,Z 499.822,A -85,B 0,C 180,E1 -3052.053,E2 -3052.053} C_VEL
LIN {X 0,Y 559.254,Z 499.825,A -85,B 0,C 180,E1 -3054.953,E2 -3054.953} C_VEL
LIN {X 0,Y 559.243,Z 499.818,A -85,B 0,C 180,E1 -3057.839,E2 -3057.839} C_VEL
LIN {X 0,Y 559.268,Z 499.819,A -85,B 0,C 180,E1 -3060.72,E2 -3060.72} C_VEL
LIN {X 0,Y 559.238,Z 499.826,A -85,B 0,C 180,E1 -3062.881,E2 -3062.881} C_VEL
LIN {X 0,Y 559.231,Z 499.819,A -85,B 0,C 180,E1 -3065.77,E2 -3065.77} C_VEL
LIN {X 0,Y 559.196,Z 499.827,A -85,B 0,C 180,E1 -3068.674,E2 -3068.674} C_VEL
LIN {X 0,Y 559.199,Z 499.826,A -85,B 0,C 180,E1 -3071.6,E2 -3071.6} C_VEL
LIN {X 0,Y 559.188,Z 499.827,A -85,B 0,C 180,E1 -3074.595,E2 -3074.595} C_VEL
LIN {X 0,Y 559.155,Z 499.832,A -85,B 0,C 180,E1 -3077.557,E2 -3077.557} C_VEL
LIN {X 0,Y 559.165,Z 499.829,A -85,B 0,C 180,E1 -3079.837,E2 -3079.837} C_VEL
LIN {X 0,Y 559.133,Z 499.832,A -85,B 0,C 180,E1 -3082.153,E2 -3082.153} C_VEL
LIN {X 0,Y 559.169,Z 499.837,A -85,B 0,C 180,E1 -3085.187,E2 -3085.187} C_VEL
LIN {X 0,Y 559.185,Z 499.829,A -85,B 0,C 180,E1 -3087.711,E2 -3087.711} C_VEL
LIN {X 0,Y 559.144,Z 499.833,A -85,B 0,C 180,E1 -3090.631,E2 -3090.631} C_VEL
LIN {X 0,Y 558.481,Z 499.923,A -85,B 0,C 180,E1 -3091.233,E2 -3091.233} C_VEL
LIN {X 0,Y 555.617,Z 500.278,A -85,B 0,C 180,E1 -3092.209,E2 -3092.209} C_VEL
LIN {X 0,Y 553.207,Z 500.578,A -85,B 0,C 180,E1 -3092.995,E2 -3092.995} C_VEL
LIN {X 0,Y 552.195,Z 500.704,A -85,B 0,C 180,E1 -3093.601,E2 -3093.601} C_VEL
LIN {X 0,Y 552.124,Z 500.71,A -85,B 0,C 180,E1 -3093.807,E2 -3093.807} C_VEL
LIN {X 0,Y 552.209,Z 500.831,A -85,B 0,C 180,E1 -3094.264,E2 -3094.264} C_VEL
LIN {X 0,Y 552.229,Z 511.812,A -85,B 0,C 180,E1 -3096.481,E2 -3096.481} C_VEL
LIN {X 0,Y 552.164,Z 517.812,A -85,B 0,C 180,E1 -3097.679,E2 -3097.679} C_VEL
LIN {X 0,Y 553.441,Z 526.677,A -85,B 0,C 180,E1 -3097.846,E2 -3097.846} C_VEL
LIN {X 0,Y 553.115,Z 623.892,A -85,B 0,C 180,E1 -3099.126,E2 -3099.126} C_VEL
LIN {X 0,Y 552.962,Z 637.737,A -85,B 0,C 180,E1 -3099.467,E2 -3099.467} C_VEL
LIN {X 0,Y 552.84,Z 650.537,A -85,B 0,C 180,E1 -3099.939,E2 -3099.939} C_VEL
LIN {X 0,Y 552.601,Z 662.763,A -85,B 0,C 180,E1 -3100.557,E2 -3100.557} C_VEL
LIN {X 0,Y 552.428,Z 674.149,A -85,B 0,C 180,E1 -3101.298,E2 -3101.298} C_VEL
LIN {X 0,Y 552.246,Z 684.808,A -85,B 0,C 180,E1 -3102.167,E2 -3102.167} C_VEL
LIN {X 0,Y 552.08,Z 694.68,A -85,B 0,C 180,E1 -3103.175,E2 -3103.175} C_VEL
LIN {X 0,Y 551.95,Z 702.828,A -85,B 0,C 180,E1 -3104.197,E2 -3104.197} C_VEL
LIN {X 0,Y 551.864,Z 709.876,A -85,B 0,C 180,E1 -3105.285,E2 -3105.285} C_VEL
LIN {X 0,Y 551.773,Z 716.319,A -85,B 0,C 180,E1 -3106.553,E2 -3106.553} C_VEL
LIN {X 0,Y 551.748,Z 720.561,A -85,B 0,C 180,E1 -3107.627,E2 -3107.627} C_VEL
LIN {X 0,Y 551.698,Z 723.851,A -85,B 0,C 180,E1 -3108.728,E2 -3108.728} C_VEL
LIN {X 0,Y 551.643,Z 726.196,A -85,B 0,C 180,E1 -3109.854,E2 -3109.854} C_VEL
LIN {X 0,Y 551.634,Z 727.581,A -85,B 0,C 180,E1 -3111.001,E2 -3111.001} C_VEL
LIN {X 0,Y 551.628,Z 727.952,A -85,B 0,C 180,E1 -3112.3,E2 -3112.3} C_VEL
LIN {X 0,Y 551.641,Z 727.319,A -85,B 0,C 180,E1 -3113.381,E2 -3113.381} C_VEL
LIN {X 0,Y 551.671,Z 725.504,A -85,B 0,C 180,E1 -3114.619,E2 -3114.619} C_VEL
LIN {X 0,Y 551.707,Z 722.337,A -85,B 0,C 180,E1 -3115.911,E2 -3115.911} C_VEL
LIN {X 0,Y 551.755,Z 717.748,A -85,B 0,C 180,E1 -3117.211,E2 -3117.211} C_VEL
LIN {X 0,Y 551.852,Z 712.602,A -85,B 0,C 180,E1 -3118.31,E2 -3118.31} C_VEL
LIN {X 0,Y 551.921,Z 705.242,A -85,B 0,C 180,E1 -3119.544,E2 -3119.544} C_VEL
LIN {X 0,Y 552.051,Z 696.962,A -85,B 0,C 180,E1 -3120.652,E2 -3120.652} C_VEL
LIN {X 0,Y 552.174,Z 688.316,A -85,B 0,C 180,E1 -3121.591,E2 -3121.591} C_VEL
LIN {X 0,Y 552.386,Z 677.525,A -85,B 0,C 180,E1 -3122.536,E2 -3122.536} C_VEL
LIN {X 0,Y 552.554,Z 666.902,A -85,B 0,C 180,E1 -3123.285,E2 -3123.285} C_VEL
LIN {X 0,Y 552.751,Z 655.271,A -85,B 0,C 180,E1 -3123.932,E2 -3123.932} C_VEL
LIN {X 0,Y 552.886,Z 643.292,A -85,B 0,C 180,E1 -3124.438,E2 -3124.438} C_VEL
LIN {X 0,Y 553.046,Z 629.714,A -85,B 0,C 180,E1 -3124.843,E2 -3124.843} C_VEL
LIN {X 0,Y 553.159,Z 615.665,A -85,B 0,C 180,E1 -3125.087,E2 -3125.087} C_VEL
LIN {X 0,Y 553.338,Z 525.006,A -85,B 0,C 180,E1 -3126.268,E2 -3126.268} C_VEL
LIN {X 0,Y 552.139,Z 517.801,A -85,B 0,C 180,E1 -3126.414,E2 -3126.414} C_VEL
LIN {X 0,Y 552.291,Z 504.268,A -85,B 0,C 180,E1 -3129.127,E2 -3129.127} C_VEL
LIN {X 0,Y 552.172,Z 500.705,A -85,B 0,C 180,E1 -3129.901,E2 -3129.901} C_VEL
LIN {X 0,Y 552.153,Z 500.71,A -85,B 0,C 180,E1 -3132.978,E2 -3132.978} C_VEL
LIN {X 0,Y 552.134,Z 500.703,A -85,B 0,C 180,E1 -3136.005,E2 -3136.005} C_VEL
LIN {X 0,Y 552.16,Z 500.708,A -85,B 0,C 180,E1 -3138.994,E2 -3138.994} C_VEL
LIN {X 0,Y 552.157,Z 500.7,A -85,B 0,C 180,E1 -3141.952,E2 -3141.952} C_VEL
LIN {X 0,Y 552.227,Z 500.701,A -85,B 0,C 180,E1 -3144.889,E2 -3144.889} C_VEL
LIN {X 0,Y 552.224,Z 500.692,A -85,B 0,C 180,E1 -3147.812,E2 -3147.812} C_VEL
LIN {X 0,Y 552.242,Z 500.696,A -85,B 0,C 180,E1 -3150.729,E2 -3150.729} C_VEL
LIN {X 0,Y 552.204,Z 500.704,A -85,B 0,C 180,E1 -3152.918,E2 -3152.918} C_VEL
LIN {X 0,Y 552.205,Z 500.694,A -85,B 0,C 180,E1 -3155.844,E2 -3155.844} C_VEL
LIN {X 0,Y 552.16,Z 500.707,A -85,B 0,C 180,E1 -3158.785,E2 -3158.785} C_VEL
LIN {X 0,Y 552.16,Z 500.7,A -85,B 0,C 180,E1 -3161.75,E2 -3161.75} C_VEL
LIN {X 0,Y 552.134,Z 500.709,A -85,B 0,C 180,E1 -3164.748,E2 -3164.748} C_VEL
LIN {X 0,Y 552.111,Z 500.706,A -85,B 0,C 180,E1 -3167.788,E2 -3167.788} C_VEL
LIN {X 0,Y 552.128,Z 500.704,A -85,B 0,C 180,E1 -3170.101,E2 -3170.101} C_VEL
LIN {X 0,Y 552.092,Z 500.71,A -85,B 0,C 180,E1 -3172.45,E2 -3172.45} C_VEL
LIN {X 0,Y 552.151,Z 500.705,A -85,B 0,C 180,E1 -3175.35,E2 -3175.35} C_VEL
LIN {X 0,Y 552.121,Z 500.704,A -85,B 0,C 180,E1 -3178.097,E2 -3178.097} C_VEL
LIN {X 0,Y 552.11,Z 500.71,A -85,B 0,C 180,E1 -3180.608,E2 -3180.608} C_VEL
LIN {X 0,Y 552.117,Z 500.712,A -85,B 0,C 180,E1 -3183.185,E2 -3183.185} C_VEL
LIN {X 0,Y 552.107,Z 500.707,A -85,B 0,C 180,E1 -3185.841,E2 -3185.841} C_VEL
LIN {X 0,Y 552.121,Z 500.715,A -85,B 0,C 180,E1 -3189.062,E2 -3189.062} C_VEL
LIN {X 0,Y 552.165,Z 500.703,A -85,B 0,C 180,E1 -3191.441,E2 -3191.441} C_VEL
LIN {X 0,Y 552.089,Z 500.711,A -85,B 0,C 180,E1 -3194.532,E2 -3194.532} C_VEL
LIN {X 0,Y 552.122,Z 500.707,A -85,B 0,C 180,E1 -3197.584,E2 -3197.584} C_VEL
LIN {X 0,Y 552.127,Z 500.705,A -85,B 0,C 180,E1 -3200.473,E2 -3200.473} C_VEL
LIN {X 0,Y 552.113,Z 500.712,A -85,B 0,C 180,E1 -3203.314,E2 -3203.314} C_VEL
LIN {X 0,Y 552.132,Z 500.703,A -85,B 0,C 180,E1 -3205.94,E2 -3205.94} C_VEL
LIN {X 0,Y 552.108,Z 500.708,A -85,B 0,C 180,E1 -3208.54,E2 -3208.54} C_VEL
LIN {X 0,Y 552.118,Z 500.71,A -85,B 0,C 180,E1 -3211.437,E2 -3211.437} C_VEL
LIN {X 0,Y 552.131,Z 500.704,A -85,B 0,C 180,E1 -3214.356,E2 -3214.356} C_VEL
LIN {X 0,Y 552.101,Z 500.711,A -85,B 0,C 180,E1 -3216.758,E2 -3216.758} C_VEL
LIN {X 0,Y 552.118,Z 500.715,A -85,B 0,C 180,E1 -3219.12,E2 -3219.12} C_VEL
LIN {X 0,Y 552.123,Z 500.709,A -85,B 0,C 180,E1 -3221.445,E2 -3221.445} C_VEL
LIN {X 0,Y 552.112,Z 500.707,A -85,B 0,C 180,E1 -3223.738,E2 -3223.738} C_VEL
LIN {X 0,Y 552.127,Z 500.704,A -85,B 0,C 180,E1 -3226.005,E2 -3226.005} C_VEL
LIN {X 0,Y 552.184,Z 500.704,A -85,B 0,C 180,E1 -3228.994,E2 -3228.994} C_VEL
LIN {X 0,Y 552.157,Z 500.7,A -85,B 0,C 180,E1 -3231.952,E2 -3231.952} C_VEL
LIN {X 0,Y 552.229,Z 500.696,A -85,B 0,C 180,E1 -3234.889,E2 -3234.889} C_VEL
LIN {X 0,Y 552.215,Z 500.694,A -85,B 0,C 180,E1 -3237.812,E2 -3237.812} C_VEL
LIN {X 0,Y 552.239,Z 500.693,A -85,B 0,C 180,E1 -3240.73,E2 -3240.73} C_VEL
LIN {X 0,Y 552.205,Z 500.699,A -85,B 0,C 180,E1 -3242.918,E2 -3242.918} C_VEL
LIN {X 0,Y 552.201,Z 500.696,A -85,B 0,C 180,E1 -3245.844,E2 -3245.844} C_VEL
LIN {X 0,Y 552.165,Z 500.702,A -85,B 0,C 180,E1 -3248.786,E2 -3248.786} C_VEL
LIN {X 0,Y 552.156,Z 500.703,A -85,B 0,C 180,E1 -3251.751,E2 -3251.751} C_VEL
LIN {X 0,Y 552.128,Z 500.706,A -85,B 0,C 180,E1 -3254.749,E2 -3254.749} C_VEL
LIN {X 0,Y 552.108,Z 500.708,A -85,B 0,C 180,E1 -3257.789,E2 -3257.789} C_VEL
LIN {X 0,Y 552.126,Z 500.704,A -85,B 0,C 180,E1 -3260.102,E2 -3260.102} C_VEL
LIN {X 0,Y 552.089,Z 500.709,A -85,B 0,C 180,E1 -3262.451,E2 -3262.451} C_VEL
LIN {X 0,Y 552.15,Z 500.71,A -85,B 0,C 180,E1 -3265.352,E2 -3265.352} C_VEL
LIN {X 0,Y 552.12,Z 500.705,A -85,B 0,C 180,E1 -3268.098,E2 -3268.098} C_VEL
LIN {X 0,Y 552.108,Z 500.707,A -85,B 0,C 180,E1 -3270.609,E2 -3270.609} C_VEL
LIN {X 0,Y 552.123,Z 500.712,A -85,B 0,C 180,E1 -3273.186,E2 -3273.186} C_VEL
LIN {X 0,Y 552.109,Z 500.708,A -85,B 0,C 180,E1 -3275.842,E2 -3275.842} C_VEL
LIN {X 0,Y 552.122,Z 500.71,A -85,B 0,C 180,E1 -3279.063,E2 -3279.063} C_VEL
LIN {X 0,Y 552.136,Z 500.711,A -85,B 0,C 180,E1 -3281.445,E2 -3281.445} C_VEL
LIN {X 0,Y 552.093,Z 500.708,A -85,B 0,C 180,E1 -3284.533,E2 -3284.533} C_VEL
LIN {X 0,Y 552.129,Z 500.71,A -85,B 0,C 180,E1 -3287.585,E2 -3287.585} C_VEL
LIN {X 0,Y 552.133,Z 500.703,A -85,B 0,C 180,E1 -3290.474,E2 -3290.474} C_VEL
LIN {X 0,Y 552.11,Z 500.715,A -85,B 0,C 180,E1 -3293.317,E2 -3293.317} C_VEL
LIN {X 0,Y 552.128,Z 500.707,A -85,B 0,C 180,E1 -3295.94,E2 -3295.94} C_VEL
LIN {X 0,Y 552.119,Z 500.706,A -85,B 0,C 180,E1 -3298.541,E2 -3298.541} C_VEL
LIN {X 0,Y 552.125,Z 500.714,A -85,B 0,C 180,E1 -3301.439,E2 -3301.439} C_VEL
LIN {X 0,Y 552.131,Z 500.708,A -85,B 0,C 180,E1 -3304.356,E2 -3304.356} C_VEL
LIN {X 0,Y 552.193,Z 500.736,A -85,B 0,C 180,E1 -3305.127,E2 -3305.127} C_VEL
LIN {X 0,Y 553.465,Z 508.024,A -85,B 0,C 180,E1 -3306.226,E2 -3306.226} C_VEL
LIN {X 0,Y 553.183,Z 526.172,A -85,B 0,C 180,E1 -3308.772,E2 -3308.772} C_VEL
LIN {X 0,Y 552.882,Z 545.419,A -85,B 0,C 180,E1 -3311.471,E2 -3311.471} C_VEL
LIN {X 0,Y 552.547,Z 565.89,A -85,B 0,C 180,E1 -3314.319,E2 -3314.319} C_VEL
LIN {X 0,Y 552.442,Z 575.357,A -85,B 0,C 180,E1 -3315.625,E2 -3315.625} C_VEL
LIN {X 0,Y 553.419,Z 583.324,A -85,B 0,C 180,E1 -3315.757,E2 -3315.757} C_VEL
LIN {X 0,Y 553.094,Z 683.962,A -85,B 0,C 180,E1 -3317.082,E2 -3317.082} C_VEL
LIN {X 0,Y 552.995,Z 697.228,A -85,B 0,C 180,E1 -3317.406,E2 -3317.406} C_VEL
LIN {X 0,Y 552.848,Z 709.376,A -85,B 0,C 180,E1 -3317.846,E2 -3317.846} C_VEL
LIN {X 0,Y 552.69,Z 721.668,A -85,B 0,C 180,E1 -3318.449,E2 -3318.449} C_VEL
LIN {X 0,Y 552.484,Z 733.201,A -85,B 0,C 180,E1 -3319.186,E2 -3319.186} C_VEL
LIN {X 0,Y 552.268,Z 743.606,A -85,B 0,C 180,E1 -3320.015,E2 -3320.015} C_VEL
LIN {X 0,Y 552.125,Z 752.115,A -85,B 0,C 180,E1 -3320.845,E2 -3320.845} C_VEL
LIN {X 0,Y 552.013,Z 759.962,A -85,B 0,C 180,E1 -3321.765,E2 -3321.765} C_VEL
LIN {X 0,Y 551.89,Z 767.622,A -85,B 0,C 180,E1 -3322.868,E2 -3322.868} C_VEL
LIN {X 0,Y 551.867,Z 774.68,A -85,B 0,C 180,E1 -3324.153,E2 -3324.153} C_VEL
LIN {X 0,Y 551.725,Z 779.373,A -85,B 0,C 180,E1 -3325.251,E2 -3325.251} C_VEL
LIN {X 0,Y 551.75,Z 782.958,A -85,B 0,C 180,E1 -3326.349,E2 -3326.349} C_VEL
LIN {X 0,Y 551.724,Z 784.808,A -85,B 0,C 180,E1 -3327.079,E2 -3327.079} C_VEL
LIN {X 0,Y 551.645,Z 787.184,A -85,B 0,C 180,E1 -3328.54,E2 -3328.54} C_VEL
LIN {X 0,Y 551.64,Z 788,A -85,B 0,C 180,E1 -3330,E2 -3330} C_VEL
LIN {X 0,Y 551.645,Z 787.185,A -85,B 0,C 180,E1 -3331.46,E2 -3331.46} C_VEL
LIN {X 0,Y 551.724,Z 784.81,A -85,B 0,C 180,E1 -3332.921,E2 -3332.921} C_VEL
LIN {X 0,Y 551.764,Z 781.896,A -85,B 0,C 180,E1 -3334.017,E2 -3334.017} C_VEL
LIN {X 0,Y 551.724,Z 777.949,A -85,B 0,C 180,E1 -3335.116,E2 -3335.116} C_VEL
LIN {X 0,Y 551.803,Z 772.192,A -85,B 0,C 180,E1 -3336.341,E2 -3336.341} C_VEL
LIN {X 0,Y 551.926,Z 765.238,A -85,B 0,C 180,E1 -3337.499,E2 -3337.499} C_VEL
LIN {X 0,Y 552.082,Z 756.993,A -85,B 0,C 180,E1 -3338.602,E2 -3338.602} C_VEL
LIN {X 0,Y 552.222,Z 748.541,A -85,B 0,C 180,E1 -3339.523,E2 -3339.523} C_VEL
LIN {X 0,Y 552.412,Z 738.098,A -85,B 0,C 180,E1 -3340.445,E2 -3340.445} C_VEL
LIN {X 0,Y 552.603,Z 727.134,A -85,B 0,C 180,E1 -3341.224,E2 -3341.224} C_VEL
LIN {X 0,Y 552.753,Z 716.413,A -85,B 0,C 180,E1 -3341.83,E2 -3341.83} C_VEL
LIN {X 0,Y 552.878,Z 704.772,A -85,B 0,C 180,E1 -3342.34,E2 -3342.34} C_VEL
LIN {X 0,Y 553.058,Z 691.358,A -85,B 0,C 180,E1 -3342.755,E2 -3342.755} C_VEL
LIN {X 0,Y 553.181,Z 678.106,A -85,B 0,C 180,E1 -3343.009,E2 -3343.009} C_VEL
LIN {X 0,Y 553.303,Z 580.888,A -85,B 0,C 180,E1 -3344.278,E2 -3344.278} C_VEL
LIN {X 0,Y 552.443,Z 575.272,A -85,B 0,C 180,E1 -3344.387,E2 -3344.387} C_VEL
LIN {X 0,Y 552.76,Z 552.597,A -85,B 0,C 180,E1 -3347.526,E2 -3347.526} C_VEL
LIN {X 0,Y 553.165,Z 530.354,A -85,B 0,C 180,E1 -3350.644,E2 -3350.644} C_VEL
LIN {X 0,Y 553.475,Z 509.493,A -85,B 0,C 180,E1 -3353.552,E2 -3353.552} C_VEL
LIN {X 0,Y 553.05,Z 505.073,A -85,B 0,C 180,E1 -3354.193,E2 -3354.193} C_VEL
LIN {X 0,Y 552.193,Z 500.705,A -85,B 0,C 180,E1 -3354.873,E2 -3354.873} C_VEL
LIN {X 0,Y 552.12,Z 500.709,A -85,B 0,C 180,E1 -3358.097,E2 -3358.097} C_VEL
LIN {X 0,Y 552.108,Z 500.716,A -85,B 0,C 180,E1 -3360.608,E2 -3360.608} C_VEL
LIN {X 0,Y 552.123,Z 500.709,A -85,B 0,C 180,E1 -3363.184,E2 -3363.184} C_VEL
LIN {X 0,Y 552.112,Z 500.707,A -85,B 0,C 180,E1 -3365.841,E2 -3365.841} C_VEL
LIN {X 0,Y 552.124,Z 500.709,A -85,B 0,C 180,E1 -3369.061,E2 -3369.061} C_VEL
LIN {X 0,Y 552.138,Z 500.704,A -85,B 0,C 180,E1 -3371.443,E2 -3371.443} C_VEL
LIN {X 0,Y 552.094,Z 500.715,A -85,B 0,C 180,E1 -3374.531,E2 -3374.531} C_VEL
LIN {X 0,Y 552.127,Z 500.703,A -85,B 0,C 180,E1 -3377.584,E2 -3377.584} C_VEL
LIN {X 0,Y 552.13,Z 500.709,A -85,B 0,C 180,E1 -3380.472,E2 -3380.472} C_VEL
LIN {X 0,Y 552.11,Z 500.708,A -85,B 0,C 180,E1 -3383.315,E2 -3383.315} C_VEL
LIN {X 0,Y 552.135,Z 500.702,A -85,B 0,C 180,E1 -3385.939,E2 -3385.939} C_VEL
LIN {X 0,Y 552.112,Z 500.712,A -85,B 0,C 180,E1 -3388.54,E2 -3388.54} C_VEL
LIN {X 0,Y 552.12,Z 500.706,A -85,B 0,C 180,E1 -3391.436,E2 -3391.436} C_VEL
LIN {X 0,Y 552.131,Z 500.706,A -85,B 0,C 180,E1 -3394.355,E2 -3394.355} C_VEL
LIN {X 0,Y 552.103,Z 500.714,A -85,B 0,C 180,E1 -3396.758,E2 -3396.758} C_VEL
LIN {X 0,Y 552.119,Z 500.71,A -85,B 0,C 180,E1 -3399.119,E2 -3399.119} C_VEL
LIN {X 0,Y 552.129,Z 500.706,A -85,B 0,C 180,E1 -3401.444,E2 -3401.444} C_VEL
LIN {X 0,Y 552.113,Z 500.706,A -85,B 0,C 180,E1 -3403.737,E2 -3403.737} C_VEL
LIN {X 0,Y 552.128,Z 500.703,A -85,B 0,C 180,E1 -3406.004,E2 -3406.004} C_VEL
LIN {X 0,Y 552.17,Z 500.707,A -85,B 0,C 180,E1 -3408.993,E2 -3408.993} C_VEL
LIN {X 0,Y 552.158,Z 500.7,A -85,B 0,C 180,E1 -3411.951,E2 -3411.951} C_VEL
LIN {X 0,Y 552.228,Z 500.699,A -85,B 0,C 180,E1 -3414.889,E2 -3414.889} C_VEL
LIN {X 0,Y 552.214,Z 500.693,A -85,B 0,C 180,E1 -3417.812,E2 -3417.812} C_VEL
LIN {X 0,Y 552.238,Z 500.695,A -85,B 0,C 180,E1 -3420.729,E2 -3420.729} C_VEL
LIN {X 0,Y 552.204,Z 500.703,A -85,B 0,C 180,E1 -3422.918,E2 -3422.918} C_VEL
LIN {X 0,Y 552.2,Z 500.695,A -85,B 0,C 180,E1 -3425.844,E2 -3425.844} C_VEL
LIN {X 0,Y 552.163,Z 500.705,A -85,B 0,C 180,E1 -3428.785,E2 -3428.785} C_VEL
LIN {X 0,Y 552.154,Z 500.702,A -85,B 0,C 180,E1 -3431.75,E2 -3431.75} C_VEL
LIN {X 0,Y 552.126,Z 500.709,A -85,B 0,C 180,E1 -3434.748,E2 -3434.748} C_VEL
LIN {X 0,Y 552.106,Z 500.708,A -85,B 0,C 180,E1 -3437.788,E2 -3437.788} C_VEL
LIN {X 0,Y 552.124,Z 500.705,A -85,B 0,C 180,E1 -3440.101,E2 -3440.101} C_VEL
LIN {X 0,Y 552.087,Z 500.711,A -85,B 0,C 180,E1 -3442.451,E2 -3442.451} C_VEL
LIN {X 0,Y 552.147,Z 500.711,A -85,B 0,C 180,E1 -3445.351,E2 -3445.351} C_VEL
LIN {X 0,Y 552.118,Z 500.707,A -85,B 0,C 180,E1 -3448.097,E2 -3448.097} C_VEL
LIN {X 0,Y 552.104,Z 500.71,A -85,B 0,C 180,E1 -3450.626,E2 -3450.626} C_VEL
LIN {X 0,Y 552.119,Z 500.715,A -85,B 0,C 180,E1 -3453.185,E2 -3453.185} C_VEL
LIN {X 0,Y 552.124,Z 500.71,A -85,B 0,C 180,E1 -3453.807,E2 -3453.807} C_VEL
LIN {X 0,Y 551.83,Z 501.262,A -85,B 0,C 180,E1 -3454.21,E2 -3454.21} C_VEL
LIN {X 0,Y 550.804,Z 503.121,A -85,B 0,C 180,E1 -3454.683,E2 -3454.683} C_VEL
LIN {X 0,Y 545.875,Z 511.223,A -85,B 0,C 180,E1 -3456.167,E2 -3456.167} C_VEL
LIN {X 0,Y 545.166,Z 513.986,A -85,B 0,C 180,E1 -3456.715,E2 -3456.715} C_VEL
LIN {X 0,Y 545.093,Z 517.879,A -85,B 0,C 180,E1 -3457.502,E2 -3457.502} C_VEL
LIN {X 0,Y 546.559,Z 527.526,A -85,B 0,C 180,E1 -3457.675,E2 -3457.675} C_VEL
LIN {X 0,Y 546.192,Z 624.42,A -85,B 0,C 180,E1 -3458.971,E2 -3458.971} C_VEL
LIN {X 0,Y 546.044,Z 637.892,A -85,B 0,C 180,E1 -3459.309,E2 -3459.309} C_VEL
LIN {X 0,Y 545.897,Z 650.057,A -85,B 0,C 180,E1 -3459.762,E2 -3459.762} C_VEL
LIN {X 0,Y 545.642,Z 662.463,A -85,B 0,C 180,E1 -3460.39,E2 -3460.39} C_VEL
LIN {X 0,Y 545.468,Z 673.044,A -85,B 0,C 180,E1 -3461.079,E2 -3461.079} C_VEL
LIN {X 0,Y 545.22,Z 683.799,A -85,B 0,C 180,E1 -3461.947,E2 -3461.947} C_VEL
LIN {X 0,Y 545.084,Z 693.077,A -85,B 0,C 180,E1 -3462.876,E2 -3462.876} C_VEL
LIN {X 0,Y 544.895,Z 701.624,A -85,B 0,C 180,E1 -3463.929,E2 -3463.929} C_VEL
LIN {X 0,Y 544.813,Z 708.88,A -85,B 0,C 180,E1 -3465.03,E2 -3465.03} C_VEL
LIN {X 0,Y 544.707,Z 715.365,A -85,B 0,C 180,E1 -3466.263,E2 -3466.263} C_VEL
LIN {X 0,Y 544.67,Z 719.804,A -85,B 0,C 180,E1 -3467.347,E2 -3467.347} C_VEL
LIN {X 0,Y 544.64,Z 723.269,A -85,B 0,C 180,E1 -3468.454,E2 -3468.454} C_VEL
LIN {X 0,Y 544.547,Z 726.177,A -85,B 0,C 180,E1 -3469.812,E2 -3469.812} C_VEL
LIN {X 0,Y 544.545,Z 727.407,A -85,B 0,C 180,E1 -3470.774,E2 -3470.774} C_VEL
LIN {X 0,Y 544.523,Z 727.983,A -85,B 0,C 180,E1 -3471.934,E2 -3471.934} C_VEL
LIN {X 0,Y 544.555,Z 727.552,A -85,B 0,C 180,E1 -3473.145,E2 -3473.145} C_VEL
LIN {X 0,Y 544.559,Z 725.806,A -85,B 0,C 180,E1 -3474.497,E2 -3474.497} C_VEL
LIN {X 0,Y 544.61,Z 723.146,A -85,B 0,C 180,E1 -3475.679,E2 -3475.679} C_VEL
LIN {X 0,Y 544.641,Z 718.792,A -85,B 0,C 180,E1 -3477.008,E2 -3477.008} C_VEL
LIN {X 0,Y 544.755,Z 714.206,A -85,B 0,C 180,E1 -3478.066,E2 -3478.066} C_VEL
LIN {X 0,Y 544.841,Z 707.022,A -85,B 0,C 180,E1 -3479.37,E2 -3479.37} C_VEL
LIN {X 0,Y 544.956,Z 699.512,A -85,B 0,C 180,E1 -3480.444,E2 -3480.444} C_VEL
LIN {X 0,Y 545.099,Z 690.317,A -85,B 0,C 180,E1 -3481.508,E2 -3481.508} C_VEL
LIN {X 0,Y 545.344,Z 679.943,A -85,B 0,C 180,E1 -3482.478,E2 -3482.478} C_VEL
LIN {X 0,Y 545.528,Z 668.851,A -85,B 0,C 180,E1 -3483.302,E2 -3483.302} C_VEL
LIN {X 0,Y 545.77,Z 656.293,A -85,B 0,C 180,E1 -3484.035,E2 -3484.035} C_VEL
LIN {X 0,Y 545.953,Z 643.697,A -85,B 0,C 180,E1 -3484.583,E2 -3484.583} C_VEL
LIN {X 0,Y 546.116,Z 630.113,A -85,B 0,C 180,E1 -3484.998,E2 -3484.998} C_VEL
LIN {X 0,Y 546.247,Z 617.346,A -85,B 0,C 180,E1 -3485.232,E2 -3485.232} C_VEL
LIN {X 0,Y 546.434,Z 525.347,A -85,B 0,C 180,E1 -3486.448,E2 -3486.448} C_VEL
LIN {X 0,Y 545.101,Z 517.85,A -85,B 0,C 180,E1 -3486.593,E2 -3486.593} C_VEL
LIN {X 0,Y 545.292,Z 504.951,A -85,B 0,C 180,E1 -3489.242,E2 -3489.242} C_VEL
LIN {X 0,Y 545.136,Z 501.582,A -85,B 0,C 180,E1 -3489.988,E2 -3489.988} C_VEL
LIN {X 0,Y 545.092,Z 501.589,A -85,B 0,C 180,E1 -3492.75,E2 -3492.75} C_VEL
LIN {X 0,Y 545.093,Z 501.58,A -85,B 0,C 180,E1 -3495.82,E2 -3495.82} C_VEL
LIN {X 0,Y 545.115,Z 501.587,A -85,B 0,C 180,E1 -3498.85,E2 -3498.85} C_VEL
LIN {X 0,Y 545.127,Z 501.576,A -85,B 0,C 180,E1 -3501.847,E2 -3501.847} C_VEL
LIN {X 0,Y 545.203,Z 501.575,A -85,B 0,C 180,E1 -3504.823,E2 -3504.823} C_VEL
LIN {X 0,Y 545.196,Z 501.567,A -85,B 0,C 180,E1 -3507.784,E2 -3507.784} C_VEL
LIN {X 0,Y 545.212,Z 501.572,A -85,B 0,C 180,E1 -3510.739,E2 -3510.739} C_VEL
LIN {X 0,Y 545.17,Z 501.58,A -85,B 0,C 180,E1 -3512.956,E2 -3512.956} C_VEL
LIN {X 0,Y 545.176,Z 501.57,A -85,B 0,C 180,E1 -3515.919,E2 -3515.919} C_VEL
LIN {X 0,Y 545.119,Z 501.586,A -85,B 0,C 180,E1 -3518.9,E2 -3518.9} C_VEL
LIN {X 0,Y 545.132,Z 501.575,A -85,B 0,C 180,E1 -3521.904,E2 -3521.904} C_VEL
LIN {X 0,Y 545.083,Z 501.591,A -85,B 0,C 180,E1 -3524.943,E2 -3524.943} C_VEL
LIN {X 0,Y 545.079,Z 501.582,A -85,B 0,C 180,E1 -3528.025,E2 -3528.025} C_VEL
LIN {X 0,Y 545.092,Z 501.582,A -85,B 0,C 180,E1 -3530.372,E2 -3530.372} C_VEL
LIN {X 0,Y 545.087,Z 501.583,A -85,B 0,C 180,E1 -3533.558,E2 -3533.558} C_VEL
LIN {X 0,Y 545.076,Z 501.582,A -85,B 0,C 180,E1 -3536,E2 -3536} C_VEL
LIN {X 0,Y 545.087,Z 501.586,A -85,B 0,C 180,E1 -3538.749,E2 -3538.749} C_VEL
LIN {X 0,Y 545.073,Z 501.584,A -85,B 0,C 180,E1 -3541.682,E2 -3541.682} C_VEL
LIN {X 0,Y 545.075,Z 501.585,A -85,B 0,C 180,E1 -3544.563,E2 -3544.563} C_VEL
LIN {X 0,Y 545.064,Z 501.589,A -85,B 0,C 180,E1 -3547.301,E2 -3547.301} C_VEL
LIN {X 0,Y 545.087,Z 501.581,A -85,B 0,C 180,E1 -3550.14,E2 -3550.14} C_VEL
LIN {X 0,Y 545.061,Z 501.588,A -85,B 0,C 180,E1 -3552.697,E2 -3552.697} C_VEL
LIN {X 0,Y 545.055,Z 501.593,A -85,B 0,C 180,E1 -3555.166,E2 -3555.166} C_VEL
LIN {X 0,Y 545.074,Z 501.583,A -85,B 0,C 180,E1 -3557.897,E2 -3557.897} C_VEL
LIN {X 0,Y 545.098,Z 501.583,A -85,B 0,C 180,E1 -3560.675,E2 -3560.675} C_VEL
LIN {X 0,Y 545.052,Z 501.587,A -85,B 0,C 180,E1 -3563.621,E2 -3563.621} C_VEL
LIN {X 0,Y 545.069,Z 501.583,A -85,B 0,C 180,E1 -3566.329,E2 -3566.329} C_VEL
LIN {X 0,Y 545.061,Z 501.591,A -85,B 0,C 180,E1 -3568.952,E2 -3568.952} C_VEL
LIN {X 0,Y 545.096,Z 501.583,A -85,B 0,C 180,E1 -3571.508,E2 -3571.508} C_VEL
LIN {X 0,Y 545.094,Z 501.581,A -85,B 0,C 180,E1 -3574.489,E2 -3574.489} C_VEL
LIN {X 0,Y 545.036,Z 501.595,A -85,B 0,C 180,E1 -3577.243,E2 -3577.243} C_VEL
LIN {X 0,Y 545.111,Z 501.579,A -85,B 0,C 180,E1 -3580.415,E2 -3580.415} C_VEL
LIN {X 0,Y 545.068,Z 501.587,A -85,B 0,C 180,E1 -3583.521,E2 -3583.521} C_VEL
LIN {X 0,Y 545.085,Z 501.582,A -85,B 0,C 180,E1 -3585.82,E2 -3585.82} C_VEL
LIN {X 0,Y 545.134,Z 501.58,A -85,B 0,C 180,E1 -3588.85,E2 -3588.85} C_VEL
LIN {X 0,Y 545.127,Z 501.577,A -85,B 0,C 180,E1 -3591.847,E2 -3591.847} C_VEL
LIN {X 0,Y 545.204,Z 501.57,A -85,B 0,C 180,E1 -3594.823,E2 -3594.823} C_VEL
LIN {X 0,Y 545.187,Z 501.57,A -85,B 0,C 180,E1 -3597.784,E2 -3597.784} C_VEL
LIN {X 0,Y 545.208,Z 501.569,A -85,B 0,C 180,E1 -3600.739,E2 -3600.739} C_VEL
LIN {X 0,Y 545.171,Z 501.576,A -85,B 0,C 180,E1 -3602.956,E2 -3602.956} C_VEL
LIN {X 0,Y 545.172,Z 501.571,A -85,B 0,C 180,E1 -3605.92,E2 -3605.92} C_VEL
LIN {X 0,Y 545.121,Z 501.581,A -85,B 0,C 180,E1 -3608.9,E2 -3608.9} C_VEL
LIN {X 0,Y 545.127,Z 501.577,A -85,B 0,C 180,E1 -3611.905,E2 -3611.905} C_VEL
LIN {X 0,Y 545.077,Z 501.587,A -85,B 0,C 180,E1 -3614.944,E2 -3614.944} C_VEL
LIN {X 0,Y 545.076,Z 501.583,A -85,B 0,C 180,E1 -3618.026,E2 -3618.026} C_VEL
LIN {X 0,Y 545.091,Z 501.58,A -85,B 0,C 180,E1 -3620.373,E2 -3620.373} C_VEL
LIN {X 0,Y 545.084,Z 501.586,A -85,B 0,C 180,E1 -3623.56,E2 -3623.56} C_VEL
LIN {X 0,Y 545.082,Z 501.582,A -85,B 0,C 180,E1 -3626.001,E2 -3626.001} C_VEL
LIN {X 0,Y 545.086,Z 501.583,A -85,B 0,C 180,E1 -3628.75,E2 -3628.75} C_VEL
LIN {X 0,Y 545.072,Z 501.587,A -85,B 0,C 180,E1 -3631.683,E2 -3631.683} C_VEL
LIN {X 0,Y 545.08,Z 501.582,A -85,B 0,C 180,E1 -3634.564,E2 -3634.564} C_VEL
LIN {X 0,Y 545.063,Z 501.594,A -85,B 0,C 180,E1 -3637.302,E2 -3637.302} C_VEL
LIN {X 0,Y 545.071,Z 501.583,A -85,B 0,C 180,E1 -3640.143,E2 -3640.143} C_VEL
LIN {X 0,Y 545.083,Z 501.587,A -85,B 0,C 180,E1 -3643.107,E2 -3643.107} C_VEL
LIN {X 0,Y 545.063,Z 501.584,A -85,B 0,C 180,E1 -3646.225,E2 -3646.225} C_VEL
LIN {X 0,Y 545.099,Z 501.582,A -85,B 0,C 180,E1 -3648.888,E2 -3648.888} C_VEL
LIN {X 0,Y 545.053,Z 501.589,A -85,B 0,C 180,E1 -3651.764,E2 -3651.764} C_VEL
LIN {X 0,Y 545.052,Z 501.585,A -85,B 0,C 180,E1 -3654.534,E2 -3654.534} C_VEL
LIN {X 0,Y 545.082,Z 501.59,A -85,B 0,C 180,E1 -3657.213,E2 -3657.213} C_VEL
LIN {X 0,Y 545.067,Z 501.589,A -85,B 0,C 180,E1 -3659.811,E2 -3659.811} C_VEL
LIN {X 0,Y 545.09,Z 501.583,A -85,B 0,C 180,E1 -3662.345,E2 -3662.345} C_VEL
LIN {X 0,Y 545.135,Z 501.741,A -85,B 0,C 180,E1 -3664.975,E2 -3664.975} C_VEL
LIN {X 0,Y 546.426,Z 508.019,A -85,B 0,C 180,E1 -3665.95,E2 -3665.95} C_VEL
LIN {X 0,Y 546.421,Z 518.715,A -85,B 0,C 180,E1 -3667.484,E2 -3667.484} C_VEL
LIN {X 0,Y 546.069,Z 538.05,A -85,B 0,C 180,E1 -3670.209,E2 -3670.209} C_VEL
LIN {X 0,Y 545.689,Z 559.066,A -85,B 0,C 180,E1 -3673.156,E2 -3673.156} C_VEL
LIN {X 0,Y 545.429,Z 575.343,A -85,B 0,C 180,E1 -3675.434,E2 -3675.434} C_VEL
LIN {X 0,Y 546.553,Z 583.945,A -85,B 0,C 180,E1 -3675.582,E2 -3675.582} C_VEL
LIN {X 0,Y 546.186,Z 683.962,A -85,B 0,C 180,E1 -3676.916,E2 -3676.916} C_VEL
LIN {X 0,Y 546.065,Z 697.227,A -85,B 0,C 180,E1 -3677.244,E2 -3677.244} C_VEL
LIN {X 0,Y 545.889,Z 710.495,A -85,B 0,C 180,E1 -3677.736,E2 -3677.736} C_VEL
LIN {X 0,Y 545.727,Z 722.371,A -85,B 0,C 180,E1 -3678.342,E2 -3678.342} C_VEL
LIN {X 0,Y 545.479,Z 734.489,A -85,B 0,C 180,E1 -3679.139,E2 -3679.139} C_VEL
LIN {X 0,Y 545.257,Z 744.649,A -85,B 0,C 180,E1 -3679.979,E2 -3679.979} C_VEL
LIN {X 0,Y 545.078,Z 753.788,A -85,B 0,C 180,E1 -3680.913,E2 -3680.913} C_VEL
LIN {X 0,Y 544.916,Z 762.69,A -85,B 0,C 180,E1 -3682.031,E2 -3682.031} C_VEL
LIN {X 0,Y 544.785,Z 769.85,A -85,B 0,C 180,E1 -3683.147,E2 -3683.147} C_VEL
LIN {X 0,Y 544.741,Z 776.366,A -85,B 0,C 180,E1 -3684.447,E2 -3684.447} C_VEL
LIN {X 0,Y 544.66,Z 780.677,A -85,B 0,C 180,E1 -3685.56,E2 -3685.56} C_VEL
LIN {X 0,Y 544.669,Z 782.958,A -85,B 0,C 180,E1 -3686.301,E2 -3686.301} C_VEL
LIN {X 0,Y 544.651,Z 784.808,A -85,B 0,C 180,E1 -3687.041,E2 -3687.041} C_VEL
LIN {X 0,Y 544.546,Z 787.184,A -85,B 0,C 180,E1 -3688.521,E2 -3688.521} C_VEL
LIN {X 0,Y 544.541,Z 788,A -85,B 0,C 180,E1 -3690,E2 -3690} C_VEL
LIN {X 0,Y 544.546,Z 787.185,A -85,B 0,C 180,E1 -3691.479,E2 -3691.479} C_VEL
LIN {X 0,Y 544.651,Z 784.81,A -85,B 0,C 180,E1 -3692.959,E2 -3692.959} C_VEL
LIN {X 0,Y 544.684,Z 781.896,A -85,B 0,C 180,E1 -3694.069,E2 -3694.069} C_VEL
LIN {X 0,Y 544.654,Z 777.949,A -85,B 0,C 180,E1 -3695.182,E2 -3695.182} C_VEL
LIN {X 0,Y 544.739,Z 772.706,A -85,B 0,C 180,E1 -3696.327,E2 -3696.327} C_VEL
LIN {X 0,Y 544.836,Z 766.468,A -85,B 0,C 180,E1 -3697.411,E2 -3697.411} C_VEL
LIN {X 0,Y 545.007,Z 758.479,A -85,B 0,C 180,E1 -3698.528,E2 -3698.528} C_VEL
LIN {X 0,Y 545.152,Z 750.336,A -85,B 0,C 180,E1 -3699.46,E2 -3699.46} C_VEL
LIN {X 0,Y 545.363,Z 740.401,A -85,B 0,C 180,E1 -3700.394,E2 -3700.394} C_VEL
LIN {X 0,Y 545.571,Z 729.543,A -85,B 0,C 180,E1 -3701.211,E2 -3701.211} C_VEL
LIN {X 0,Y 545.762,Z 718.178,A -85,B 0,C 180,E1 -3701.89,E2 -3701.89} C_VEL
LIN {X 0,Y 545.912,Z 705.982,A -85,B 0,C 180,E1 -3702.453,E2 -3702.453} C_VEL
LIN {X 0,Y 546.103,Z 693.186,A -85,B 0,C 180,E1 -3702.873,E2 -3702.873} C_VEL
LIN {X 0,Y 546.266,Z 679.621,A -85,B 0,C 180,E1 -3703.153,E2 -3703.153} C_VEL
LIN {X 0,Y 546.49,Z 582.167,A -85,B 0,C 180,E1 -3704.443,E2 -3704.443} C_VEL
LIN {X 0,Y 545.439,Z 575.244,A -85,B 0,C 180,E1 -3704.579,E2 -3704.579} C_VEL
LIN {X 0,Y 545.801,Z 554.203,A -85,B 0,C 180,E1 -3707.529,E2 -3707.529} C_VEL
LIN {X 0,Y 546.202,Z 531.35,A -85,B 0,C 180,E1 -3710.722,E2 -3710.722} C_VEL
LIN {X 0,Y 546.522,Z 509.83,A -85,B 0,C 180,E1 -3713.763,E2 -3713.763} C_VEL
LIN {X 0,Y 545.438,Z 503.277,A -85,B 0,C 180,E1 -3714.756,E2 -3714.756} C_VEL
LIN {X 0,Y 545.134,Z 501.583,A -85,B 0,C 180,E1 -3715.025,E2 -3715.025} C_VEL
LIN {X 0,Y 545.09,Z 501.583,A -85,B 0,C 180,E1 -3717.655,E2 -3717.655} C_VEL
LIN {X 0,Y 545.077,Z 501.588,A -85,B 0,C 180,E1 -3720.246,E2 -3720.246} C_VEL
LIN {X 0,Y 545.089,Z 501.587,A -85,B 0,C 180,E1 -3723.063,E2 -3723.063} C_VEL
LIN {X 0,Y 545.062,Z 501.586,A -85,B 0,C 180,E1 -3725.676,E2 -3725.676} C_VEL
LIN {X 0,Y 545.053,Z 501.589,A -85,B 0,C 180,E1 -3728.236,E2 -3728.236} C_VEL
LIN {X 0,Y 545.099,Z 501.584,A -85,B 0,C 180,E1 -3731.112,E2 -3731.112} C_VEL
LIN {X 0,Y 545.056,Z 501.587,A -85,B 0,C 180,E1 -3734.128,E2 -3734.128} C_VEL
LIN {X 0,Y 545.083,Z 501.588,A -85,B 0,C 180,E1 -3736.893,E2 -3736.893} C_VEL
LIN {X 0,Y 545.071,Z 501.583,A -85,B 0,C 180,E1 -3739.857,E2 -3739.857} C_VEL
LIN {X 0,Y 545.07,Z 501.588,A -85,B 0,C 180,E1 -3743.072,E2 -3743.072} C_VEL
LIN {X 0,Y 545.085,Z 501.581,A -85,B 0,C 180,E1 -3745.604,E2 -3745.604} C_VEL
LIN {X 0,Y 545.072,Z 501.586,A -85,B 0,C 180,E1 -3748.317,E2 -3748.317} C_VEL
LIN {X 0,Y 545.086,Z 501.584,A -85,B 0,C 180,E1 -3751.25,E2 -3751.25} C_VEL
LIN {X 0,Y 545.083,Z 501.582,A -85,B 0,C 180,E1 -3753.999,E2 -3753.999} C_VEL
LIN {X 0,Y 545.084,Z 501.583,A -85,B 0,C 180,E1 -3756.44,E2 -3756.44} C_VEL
LIN {X 0,Y 545.091,Z 501.58,A -85,B 0,C 180,E1 -3759.627,E2 -3759.627} C_VEL
LIN {X 0,Y 545.087,Z 501.588,A -85,B 0,C 180,E1 -3762.749,E2 -3762.749} C_VEL
LIN {X 0,Y 545.086,Z 501.581,A -85,B 0,C 180,E1 -3765.819,E2 -3765.819} C_VEL
LIN {X 0,Y 545.124,Z 501.585,A -85,B 0,C 180,E1 -3768.849,E2 -3768.849} C_VEL
LIN {X 0,Y 545.127,Z 501.576,A -85,B 0,C 180,E1 -3771.847,E2 -3771.847} C_VEL
LIN {X 0,Y 545.204,Z 501.573,A -85,B 0,C 180,E1 -3774.823,E2 -3774.823} C_VEL
LIN {X 0,Y 545.186,Z 501.569,A -85,B 0,C 180,E1 -3777.783,E2 -3777.783} C_VEL
LIN {X 0,Y 545.208,Z 501.571,A -85,B 0,C 180,E1 -3780.738,E2 -3780.738} C_VEL
LIN {X 0,Y 545.17,Z 501.58,A -85,B 0,C 180,E1 -3782.955,E2 -3782.955} C_VEL
LIN {X 0,Y 545.171,Z 501.57,A -85,B 0,C 180,E1 -3785.919,E2 -3785.919} C_VEL
LIN {X 0,Y 545.12,Z 501.584,A -85,B 0,C 180,E1 -3788.9,E2 -3788.9} C_VEL
LIN {X 0,Y 545.126,Z 501.577,A -85,B 0,C 180,E1 -3791.904,E2 -3791.904} C_VEL
LIN {X 0,Y 545.075,Z 501.59,A -85,B 0,C 180,E1 -3794.943,E2 -3794.943} C_VEL
LIN {X 0,Y 545.075,Z 501.583,A -85,B 0,C 180,E1 -3798.025,E2 -3798.025} C_VEL
LIN {X 0,Y 545.089,Z 501.582,A -85,B 0,C 180,E1 -3800.372,E2 -3800.372} C_VEL
LIN {X 0,Y 545.081,Z 501.588,A -85,B 0,C 180,E1 -3803.559,E2 -3803.559} C_VEL
LIN {X 0,Y 545.08,Z 501.585,A -85,B 0,C 180,E1 -3806,E2 -3806} C_VEL
LIN {X 0,Y 545.084,Z 501.587,A -85,B 0,C 180,E1 -3808.749,E2 -3808.749} C_VEL
LIN {X 0,Y 545.068,Z 501.59,A -85,B 0,C 180,E1 -3811.683,E2 -3811.683} C_VEL
LIN {X 0,Y 545.157,Z 501.73,A -85,B 0,C 180,E1 -3814.151,E2 -3814.151} C_VEL
LIN {X 0,Y 545.222,Z 510.48,A -85,B 0,C 180,E1 -3816.003,E2 -3816.003} C_VEL
LIN {X 0,Y 545.166,Z 513.986,A -85,B 0,C 180,E1 -3816.715,E2 -3816.715} C_VEL
LIN {X 0,Y 544.882,Z 516.312,A -85,B 0,C 180,E1 -3817.029,E2 -3817.029} C_VEL
LIN {X 0,Y 544.244,Z 519.39,A -85,B 0,C 180,E1 -3817.26,E2 -3817.26} C_VEL
LIN {X 0,Y 542.935,Z 524.777,A -85,B 0,C 180,E1 -3817.481,E2 -3817.481} C_VEL
LIN {X 0,Y 541.436,Z 530.805,A -85,B 0,C 180,E1 -3817.58,E2 -3817.58} C_VEL
LIN {X 0,Y 539.906,Z 539.246,A -85,B 0,C 180,E1 -3817.651,E2 -3817.651} C_VEL
LIN {X 0,Y 539.645,Z 543.512,A -85,B 0,C 180,E1 -3817.701,E2 -3817.701} C_VEL
LIN {X 0,Y 539.302,Z 624.136,A -85,B 0,C 180,E1 -3818.795,E2 -3818.795} C_VEL
LIN {X 0,Y 539.093,Z 637.901,A -85,B 0,C 180,E1 -3819.143,E2 -3819.143} C_VEL
LIN {X 0,Y 538.94,Z 650.715,A -85,B 0,C 180,E1 -3819.63,E2 -3819.63} C_VEL
LIN {X 0,Y 538.652,Z 663.335,A -85,B 0,C 180,E1 -3820.29,E2 -3820.29} C_VEL
LIN {X 0,Y 538.456,Z 673.863,A -85,B 0,C 180,E1 -3820.995,E2 -3820.995} C_VEL
LIN {X 0,Y 538.182,Z 684.72,A -85,B 0,C 180,E1 -3821.898,E2 -3821.898} C_VEL
LIN {X 0,Y 538.032,Z 693.33,A -85,B 0,C 180,E1 -3822.784,E2 -3822.784} C_VEL
LIN {X 0,Y 537.831,Z 701.709,A -85,B 0,C 180,E1 -3823.833,E2 -3823.833} C_VEL
LIN {X 0,Y 537.725,Z 708.613,A -85,B 0,C 180,E1 -3824.891,E2 -3824.891} C_VEL
LIN {X 0,Y 537.647,Z 715.189,A -85,B 0,C 180,E1 -3826.149,E2 -3826.149} C_VEL
LIN {X 0,Y 537.6,Z 719.385,A -85,B 0,C 180,E1 -3827.174,E2 -3827.174} C_VEL
LIN {X 0,Y 537.527,Z 723.946,A -85,B 0,C 180,E1 -3828.681,E2 -3828.681} C_VEL
LIN {X 0,Y 537.428,Z 726.726,A -85,B 0,C 180,E1 -3830.151,E2 -3830.151} C_VEL
LIN {X 0,Y 537.422,Z 727.93,A -85,B 0,C 180,E1 -3831.686,E2 -3831.686} C_VEL
LIN {X 0,Y 537.446,Z 727.64,A -85,B 0,C 180,E1 -3833.022,E2 -3833.022} C_VEL
LIN {X 0,Y 537.441,Z 726.379,A -85,B 0,C 180,E1 -3834.17,E2 -3834.17} C_VEL
LIN {X 0,Y 537.505,Z 723.823,A -85,B 0,C 180,E1 -3835.46,E2 -3835.46} C_VEL
LIN {X 0,Y 537.564,Z 719.841,A -85,B 0,C 180,E1 -3836.795,E2 -3836.795} C_VEL
LIN {X 0,Y 537.68,Z 714.096,A -85,B 0,C 180,E1 -3838.169,E2 -3838.169} C_VEL
LIN {X 0,Y 537.756,Z 707.672,A -85,B 0,C 180,E1 -3839.357,E2 -3839.357} C_VEL
LIN {X 0,Y 537.886,Z 700.338,A -85,B 0,C 180,E1 -3840.447,E2 -3840.447} C_VEL
LIN {X 0,Y 538.061,Z 691.311,A -85,B 0,C 180,E1 -3841.527,E2 -3841.527} C_VEL
LIN {X 0,Y 538.299,Z 681.41,A -85,B 0,C 180,E1 -3842.487,E2 -3842.487} C_VEL
LIN {X 0,Y 538.529,Z 670.405,A -85,B 0,C 180,E1 -3843.346,E2 -3843.346} C_VEL
LIN {X 0,Y 538.755,Z 659.433,A -85,B 0,C 180,E1 -3844.024,E2 -3844.024} C_VEL
LIN {X 0,Y 538.951,Z 647.053,A -85,B 0,C 180,E1 -3844.616,E2 -3844.616} C_VEL
LIN {X 0,Y 539.215,Z 634.363,A -85,B 0,C 180,E1 -3845.055,E2 -3845.055} C_VEL
LIN {X 0,Y 539.313,Z 622.219,A -85,B 0,C 180,E1 -3845.329,E2 -3845.329} C_VEL
LIN {X 0,Y 539.602,Z 526.418,A -85,B 0,C 180,E1 -3846.62,E2 -3846.62} C_VEL
LIN {X 0,Y 538.09,Z 518.05,A -85,B 0,C 180,E1 -3846.78,E2 -3846.78} C_VEL
LIN {X 0,Y 538.295,Z 505.788,A -85,B 0,C 180,E1 -3849.359,E2 -3849.359} C_VEL
LIN {X 0,Y 538.091,Z 502.46,A -85,B 0,C 180,E1 -3850.084,E2 -3850.084} C_VEL
LIN {X 0,Y 538.022,Z 502.465,A -85,B 0,C 180,E1 -3853.299,E2 -3853.299} C_VEL
LIN {X 0,Y 538.061,Z 502.457,A -85,B 0,C 180,E1 -3855.631,E2 -3855.631} C_VEL
LIN {X 0,Y 538.074,Z 502.461,A -85,B 0,C 180,E1 -3858.702,E2 -3858.702} C_VEL
LIN {X 0,Y 538.084,Z 502.453,A -85,B 0,C 180,E1 -3861.74,E2 -3861.74} C_VEL
LIN {X 0,Y 538.161,Z 502.451,A -85,B 0,C 180,E1 -3864.755,E2 -3864.755} C_VEL
LIN {X 0,Y 538.167,Z 502.443,A -85,B 0,C 180,E1 -3867.755,E2 -3867.755} C_VEL
LIN {X 0,Y 538.182,Z 502.448,A -85,B 0,C 180,E1 -3870.748,E2 -3870.748} C_VEL
LIN {X 0,Y 538.137,Z 502.455,A -85,B 0,C 180,E1 -3872.994,E2 -3872.994} C_VEL
LIN {X 0,Y 538.13,Z 502.447,A -85,B 0,C 180,E1 -3875.997,E2 -3875.997} C_VEL
LIN {X 0,Y 538.069,Z 502.464,A -85,B 0,C 180,E1 -3879.017,E2 -3879.017} C_VEL
LIN {X 0,Y 538.081,Z 502.454,A -85,B 0,C 180,E1 -3882.062,E2 -3882.062} C_VEL
LIN {X 0,Y 538.043,Z 502.465,A -85,B 0,C 180,E1 -3885.143,E2 -3885.143} C_VEL
LIN {X 0,Y 538.031,Z 502.461,A -85,B 0,C 180,E1 -3888.27,E2 -3888.27} C_VEL
LIN {X 0,Y 538.036,Z 502.464,A -85,B 0,C 180,E1 -3890.651,E2 -3890.651} C_VEL
LIN {X 0,Y 538.02,Z 502.461,A -85,B 0,C 180,E1 -3893.887,E2 -3893.887} C_VEL
LIN {X 0,Y 538.038,Z 502.46,A -85,B 0,C 180,E1 -3896.366,E2 -3896.366} C_VEL
LIN {X 0,Y 538.051,Z 502.466,A -85,B 0,C 180,E1 -3898.938,E2 -3898.938} C_VEL
LIN {X 0,Y 538.022,Z 502.461,A -85,B 0,C 180,E1 -3901.89,E2 -3901.89} C_VEL
LIN {X 0,Y 538.025,Z 502.464,A -85,B 0,C 180,E1 -3904.62,E2 -3904.62} C_VEL
LIN {X 0,Y 538.02,Z 502.469,A -85,B 0,C 180,E1 -3907.173,E2 -3907.173} C_VEL
LIN {X 0,Y 538.049,Z 502.458,A -85,B 0,C 180,E1 -3909.794,E2 -3909.794} C_VEL
LIN {X 0,Y 538.019,Z 502.467,A -85,B 0,C 180,E1 -3912.785,E2 -3912.785} C_VEL
LIN {X 0,Y 538.021,Z 502.461,A -85,B 0,C 180,E1 -3915.925,E2 -3915.925} C_VEL
LIN {X 0,Y 538.07,Z 502.462,A -85,B 0,C 180,E1 -3919.249,E2 -3919.249} C_VEL
LIN {X 0,Y 537.994,Z 502.464,A -85,B 0,C 180,E1 -3922.123,E2 -3922.123} C_VEL
LIN {X 0,Y 538.013,Z 502.469,A -85,B 0,C 180,E1 -3924.917,E2 -3924.917} C_VEL
LIN {X 0,Y 538.022,Z 502.463,A -85,B 0,C 180,E1 -3927.618,E2 -3927.618} C_VEL
LIN {X 0,Y 538.034,Z 502.46,A -85,B 0,C 180,E1 -3930.24,E2 -3930.24} C_VEL
LIN {X 0,Y 538.062,Z 502.461,A -85,B 0,C 180,E1 -3932.797,E2 -3932.797} C_VEL
LIN {X 0,Y 538.045,Z 502.465,A -85,B 0,C 180,E1 -3935.293,E2 -3935.293} C_VEL
LIN {X 0,Y 538.005,Z 502.463,A -85,B 0,C 180,E1 -3938.042,E2 -3938.042} C_VEL
LIN {X 0,Y 538.032,Z 502.466,A -85,B 0,C 180,E1 -3940.94,E2 -3940.94} C_VEL
LIN {X 0,Y 538.019,Z 502.469,A -85,B 0,C 180,E1 -3943.299,E2 -3943.299} C_VEL
LIN {X 0,Y 538.054,Z 502.46,A -85,B 0,C 180,E1 -3945.631,E2 -3945.631} C_VEL
LIN {X 0,Y 538.087,Z 502.456,A -85,B 0,C 180,E1 -3948.702,E2 -3948.702} C_VEL
LIN {X 0,Y 538.083,Z 502.455,A -85,B 0,C 180,E1 -3951.74,E2 -3951.74} C_VEL
LIN {X 0,Y 538.18,Z 502.444,A -85,B 0,C 180,E1 -3954.756,E2 -3954.756} C_VEL
LIN {X 0,Y 538.159,Z 502.446,A -85,B 0,C 180,E1 -3957.755,E2 -3957.755} C_VEL
LIN {X 0,Y 538.178,Z 502.444,A -85,B 0,C 180,E1 -3960.749,E2 -3960.749} C_VEL
LIN {X 0,Y 538.137,Z 502.453,A -85,B 0,C 180,E1 -3962.995,E2 -3962.995} C_VEL
LIN {X 0,Y 538.125,Z 502.448,A -85,B 0,C 180,E1 -3965.998,E2 -3965.998} C_VEL
LIN {X 0,Y 538.07,Z 502.461,A -85,B 0,C 180,E1 -3969.018,E2 -3969.018} C_VEL
LIN {X 0,Y 538.076,Z 502.454,A -85,B 0,C 180,E1 -3972.063,E2 -3972.063} C_VEL
LIN {X 0,Y 538.037,Z 502.467,A -85,B 0,C 180,E1 -3975.144,E2 -3975.144} C_VEL
LIN {X 0,Y 538.028,Z 502.46,A -85,B 0,C 180,E1 -3978.271,E2 -3978.271} C_VEL
LIN {X 0,Y 538.035,Z 502.461,A -85,B 0,C 180,E1 -3980.652,E2 -3980.652} C_VEL
LIN {X 0,Y 538.016,Z 502.463,A -85,B 0,C 180,E1 -3983.888,E2 -3983.888} C_VEL
LIN {X 0,Y 538.044,Z 502.458,A -85,B 0,C 180,E1 -3986.367,E2 -3986.367} C_VEL
LIN {X 0,Y 538.05,Z 502.462,A -85,B 0,C 180,E1 -3988.939,E2 -3988.939} C_VEL
LIN {X 0,Y 538.021,Z 502.463,A -85,B 0,C 180,E1 -3991.891,E2 -3991.891} C_VEL
LIN {X 0,Y 538.03,Z 502.461,A -85,B 0,C 180,E1 -3994.622,E2 -3994.622} C_VEL
LIN {X 0,Y 538.018,Z 502.469,A -85,B 0,C 180,E1 -3997.174,E2 -3997.174} C_VEL
LIN {X 0,Y 538.026,Z 502.463,A -85,B 0,C 180,E1 -3999.797,E2 -3999.797} C_VEL
LIN {X 0,Y 538.02,Z 502.463,A -85,B 0,C 180,E1 -4002.786,E2 -4002.786} C_VEL
LIN {X 0,Y 538.027,Z 502.462,A -85,B 0,C 180,E1 -4005.926,E2 -4005.926} C_VEL
LIN {X 0,Y 538.076,Z 502.462,A -85,B 0,C 180,E1 -4009.25,E2 -4009.25} C_VEL
LIN {X 0,Y 537.993,Z 502.465,A -85,B 0,C 180,E1 -4012.123,E2 -4012.123} C_VEL
LIN {X 0,Y 538.011,Z 502.465,A -85,B 0,C 180,E1 -4014.918,E2 -4014.918} C_VEL
LIN {X 0,Y 538.031,Z 502.467,A -85,B 0,C 180,E1 -4017.619,E2 -4017.619} C_VEL
LIN {X 0,Y 538.019,Z 502.464,A -85,B 0,C 180,E1 -4020.24,E2 -4020.24} C_VEL
LIN {X 0,Y 538.064,Z 502.46,A -85,B 0,C 180,E1 -4022.797,E2 -4022.797} C_VEL
LIN {X 0,Y 538.102,Z 502.488,A -85,B 0,C 180,E1 -4024.78,E2 -4024.78} C_VEL
LIN {X 0,Y 539.536,Z 509.763,A -85,B 0,C 180,E1 -4025.924,E2 -4025.924} C_VEL
LIN {X 0,Y 539.407,Z 522.694,A -85,B 0,C 180,E1 -4027.8,E2 -4027.8} C_VEL
LIN {X 0,Y 539.025,Z 540.819,A -85,B 0,C 180,E1 -4030.383,E2 -4030.383} C_VEL
LIN {X 0,Y 538.656,Z 561.67,A -85,B 0,C 180,E1 -4033.32,E2 -4033.32} C_VEL
LIN {X 0,Y 538.455,Z 575.487,A -85,B 0,C 180,E1 -4035.246,E2 -4035.246} C_VEL
LIN {X 0,Y 539.677,Z 583.858,A -85,B 0,C 180,E1 -4035.393,E2 -4035.393} C_VEL
LIN {X 0,Y 539.284,Z 683.961,A -85,B 0,C 180,E1 -4036.745,E2 -4036.745} C_VEL
LIN {X 0,Y 539.157,Z 697.227,A -85,B 0,C 180,E1 -4037.078,E2 -4037.078} C_VEL
LIN {X 0,Y 538.951,Z 709.376,A -85,B 0,C 180,E1 -4037.527,E2 -4037.527} C_VEL
LIN {X 0,Y 538.788,Z 720.793,A -85,B 0,C 180,E1 -4038.096,E2 -4038.096} C_VEL
LIN {X 0,Y 538.535,Z 731.906,A -85,B 0,C 180,E1 -4038.807,E2 -4038.807} C_VEL
LIN {X 0,Y 538.266,Z 742.539,A -85,B 0,C 180,E1 -4039.658,E2 -4039.658} C_VEL
LIN {X 0,Y 538.067,Z 752.115,A -85,B 0,C 180,E1 -4040.604,E2 -4040.604} C_VEL
LIN {X 0,Y 537.921,Z 759.962,A -85,B 0,C 180,E1 -4041.548,E2 -4041.548} C_VEL
LIN {X 0,Y 537.755,Z 767.623,A -85,B 0,C 180,E1 -4042.679,E2 -4042.679} C_VEL
LIN {X 0,Y 537.693,Z 774.68,A -85,B 0,C 180,E1 -4043.998,E2 -4043.998} C_VEL
LIN {X 0,Y 537.541,Z 779.373,A -85,B 0,C 180,E1 -4045.125,E2 -4045.125} C_VEL
LIN {X 0,Y 537.591,Z 782.958,A -85,B 0,C 180,E1 -4046.252,E2 -4046.252} C_VEL
LIN {X 0,Y 537.551,Z 784.807,A -85,B 0,C 180,E1 -4047.002,E2 -4047.002} C_VEL
LIN {X 0,Y 537.451,Z 787.183,A -85,B 0,C 180,E1 -4048.501,E2 -4048.501} C_VEL
LIN {X 0,Y 537.442,Z 788,A -85,B 0,C 180,E1 -4050,E2 -4050} C_VEL
LIN {X 0,Y 537.451,Z 787.184,A -85,B 0,C 180,E1 -4051.499,E2 -4051.499} C_VEL
LIN {X 0,Y 537.551,Z 784.81,A -85,B 0,C 180,E1 -4052.998,E2 -4052.998} C_VEL
LIN {X 0,Y 537.603,Z 781.896,A -85,B 0,C 180,E1 -4054.123,E2 -4054.123} C_VEL
LIN {X 0,Y 537.588,Z 777.949,A -85,B 0,C 180,E1 -4055.25,E2 -4055.25} C_VEL
LIN {X 0,Y 537.65,Z 773.083,A -85,B 0,C 180,E1 -4056.335,E2 -4056.335} C_VEL
LIN {X 0,Y 537.791,Z 766.468,A -85,B 0,C 180,E1 -4057.509,E2 -4057.509} C_VEL
LIN {X 0,Y 537.972,Z 758.479,A -85,B 0,C 180,E1 -4058.64,E2 -4058.64} C_VEL
LIN {X 0,Y 538.143,Z 750.336,A -85,B 0,C 180,E1 -4059.585,E2 -4059.585} C_VEL
LIN {X 0,Y 538.352,Z 740.401,A -85,B 0,C 180,E1 -4060.531,E2 -4060.531} C_VEL
LIN {X 0,Y 538.578,Z 730.595,A -85,B 0,C 180,E1 -4061.288,E2 -4061.288} C_VEL
LIN {X 0,Y 538.804,Z 719.707,A -85,B 0,C 180,E1 -4061.963,E2 -4061.963} C_VEL
LIN {X 0,Y 538.953,Z 707.109,A -85,B 0,C 180,E1 -4062.568,E2 -4062.568} C_VEL
LIN {X 0,Y 539.188,Z 694.098,A -85,B 0,C 180,E1 -4063.017,E2 -4063.017} C_VEL
LIN {X 0,Y 539.364,Z 681.124,A -85,B 0,C 180,E1 -4063.301,E2 -4063.301} C_VEL
LIN {X 0,Y 539.614,Z 582.883,A -85,B 0,C 180,E1 -4064.622,E2 -4064.622} C_VEL
LIN {X 0,Y 538.456,Z 575.199,A -85,B 0,C 180,E1 -4064.779,E2 -4064.779} C_VEL
LIN {X 0,Y 538.805,Z 552.565,A -85,B 0,C 180,E1 -4067.952,E2 -4067.952} C_VEL
LIN {X 0,Y 539.206,Z 530.943,A -85,B 0,C 180,E1 -4071.004,E2 -4071.004} C_VEL
LIN {X 0,Y 539.587,Z 512.715,A -85,B 0,C 180,E1 -4073.61,E2 -4073.61} C_VEL
LIN {X 0,Y 539.326,Z 508.816,A -85,B 0,C 180,E1 -4074.192,E2 -4074.192} C_VEL
LIN {X 0,Y 538.102,Z 502.458,A -85,B 0,C 180,E1 -4075.22,E2 -4075.22} C_VEL
LIN {X 0,Y 538.045,Z 502.463,A -85,B 0,C 180,E1 -4078.049,E2 -4078.049} C_VEL
LIN {X 0,Y 538.021,Z 502.471,A -85,B 0,C 180,E1 -4080.626,E2 -4080.626} C_VEL
LIN {X 0,Y 538.045,Z 502.462,A -85,B 0,C 180,E1 -4083.282,E2 -4083.282} C_VEL
LIN {X 0,Y 538.027,Z 502.463,A -85,B 0,C 180,E1 -4086.001,E2 -4086.001} C_VEL
LIN {X 0,Y 538.014,Z 502.47,A -85,B 0,C 180,E1 -4088.829,E2 -4088.829} C_VEL
LIN {X 0,Y 538.076,Z 502.463,A -85,B 0,C 180,E1 -4090.772,E2 -4090.772} C_VEL
LIN {X 0,Y 538.027,Z 502.462,A -85,B 0,C 180,E1 -4094.074,E2 -4094.074} C_VEL
LIN {X 0,Y 538.02,Z 502.463,A -85,B 0,C 180,E1 -4097.214,E2 -4097.214} C_VEL
LIN {X 0,Y 538.026,Z 502.463,A -85,B 0,C 180,E1 -4100.203,E2 -4100.203} C_VEL
LIN {X 0,Y 538.025,Z 502.466,A -85,B 0,C 180,E1 -4103.067,E2 -4103.067} C_VEL
LIN {X 0,Y 538.027,Z 502.46,A -85,B 0,C 180,E1 -4105.827,E2 -4105.827} C_VEL
LIN {X 0,Y 538.018,Z 502.467,A -85,B 0,C 180,E1 -4108.499,E2 -4108.499} C_VEL
LIN {X 0,Y 538.053,Z 502.462,A -85,B 0,C 180,E1 -4111.099,E2 -4111.099} C_VEL
LIN {X 0,Y 538.044,Z 502.459,A -85,B 0,C 180,E1 -4113.633,E2 -4113.633} C_VEL
LIN {X 0,Y 538.015,Z 502.461,A -85,B 0,C 180,E1 -4116.117,E2 -4116.117} C_VEL
LIN {X 0,Y 538.035,Z 502.462,A -85,B 0,C 180,E1 -4119.348,E2 -4119.348} C_VEL
LIN {X 0,Y 538.064,Z 502.46,A -85,B 0,C 180,E1 -4122.517,E2 -4122.517} C_VEL
LIN {X 0,Y 538.055,Z 502.457,A -85,B 0,C 180,E1 -4125.63,E2 -4125.63} C_VEL
LIN {X 0,Y 538.081,Z 502.46,A -85,B 0,C 180,E1 -4128.701,E2 -4128.701} C_VEL
LIN {X 0,Y 538.083,Z 502.454,A -85,B 0,C 180,E1 -4131.739,E2 -4131.739} C_VEL
LIN {X 0,Y 538.18,Z 502.446,A -85,B 0,C 180,E1 -4134.755,E2 -4134.755} C_VEL
LIN {X 0,Y 538.158,Z 502.445,A -85,B 0,C 180,E1 -4137.754,E2 -4137.754} C_VEL
LIN {X 0,Y 538.177,Z 502.447,A -85,B 0,C 180,E1 -4140.748,E2 -4140.748} C_VEL
LIN {X 0,Y 538.136,Z 502.456,A -85,B 0,C 180,E1 -4142.994,E2 -4142.994} C_VEL
LIN {X 0,Y 538.125,Z 502.448,A -85,B 0,C 180,E1 -4145.997,E2 -4145.997} C_VEL
LIN {X 0,Y 538.069,Z 502.464,A -85,B 0,C 180,E1 -4149.017,E2 -4149.017} C_VEL
LIN {X 0,Y 538.074,Z 502.455,A -85,B 0,C 180,E1 -4152.062,E2 -4152.062} C_VEL
LIN {X 0,Y 538.036,Z 502.469,A -85,B 0,C 180,E1 -4155.144,E2 -4155.144} C_VEL
LIN {X 0,Y 538.028,Z 502.461,A -85,B 0,C 180,E1 -4158.27,E2 -4158.27} C_VEL
LIN {X 0,Y 538.033,Z 502.463,A -85,B 0,C 180,E1 -4160.651,E2 -4160.651} C_VEL
LIN {X 0,Y 538.014,Z 502.465,A -85,B 0,C 180,E1 -4163.887,E2 -4163.887} C_VEL
LIN {X 0,Y 538.041,Z 502.462,A -85,B 0,C 180,E1 -4166.366,E2 -4166.366} C_VEL
LIN {X 0,Y 538.046,Z 502.466,A -85,B 0,C 180,E1 -4168.939,E2 -4168.939} C_VEL
LIN {X 0,Y 538.018,Z 502.466,A -85,B 0,C 180,E1 -4171.891,E2 -4171.891} C_VEL
LIN {X 0,Y 538.088,Z 502.563,A -85,B 0,C 180,E1 -4174.012,E2 -4174.012} C_VEL
LIN {X 0,Y 538.317,Z 508.479,A -85,B 0,C 180,E1 -4175.28,E2 -4175.28} C_VEL
LIN {X 0,Y 538.109,Z 518.053,A -85,B 0,C 180,E1 -4177.304,E2 -4177.304} C_VEL
LIN {X 0,Y 539.677,Z 527.461,A -85,B 0,C 180,E1 -4177.486,E2 -4177.486} C_VEL
LIN {X 0,Y 539.645,Z 543.512,A -85,B 0,C 180,E1 -4177.701,E2 -4177.701} C_VEL
LIN {X 0,Y 538.921,Z 549.356,A -85,B 0,C 180,E1 -4177.76,E2 -4177.76} C_VEL
LIN {X 0,Y 533.317,Z 568.362,A -85,B 0,C 180,E1 -4177.862,E2 -4177.862} C_VEL
LIN {X 0,Y 532.642,Z 574.205,A -85,B 0,C 180,E1 -4177.923,E2 -4177.923} C_VEL
LIN {X 0,Y 532.406,Z 624.535,A -85,B 0,C 180,E1 -4178.624,E2 -4178.624} C_VEL
LIN {X 0,Y 532.19,Z 637.814,A -85,B 0,C 180,E1 -4178.963,E2 -4178.963} C_VEL
LIN {X 0,Y 532.029,Z 650.837,A -85,B 0,C 180,E1 -4179.462,E2 -4179.462} C_VEL
LIN {X 0,Y 531.782,Z 662.031,A -85,B 0,C 180,E1 -4180.045,E2 -4180.045} C_VEL
LIN {X 0,Y 531.495,Z 672.812,A -85,B 0,C 180,E1 -4180.759,E2 -4180.759} C_VEL
LIN {X 0,Y 531.193,Z 683.783,A -85,B 0,C 180,E1 -4181.669,E2 -4181.669} C_VEL
LIN {X 0,Y 531.014,Z 693.275,A -85,B 0,C 180,E1 -4182.654,E2 -4182.654} C_VEL
LIN {X 0,Y 530.77,Z 702.306,A -85,B 0,C 180,E1 -4183.808,E2 -4183.808} C_VEL
LIN {X 0,Y 530.645,Z 709.785,A -85,B 0,C 180,E1 -4184.997,E2 -4184.997} C_VEL
LIN {X 0,Y 530.581,Z 715.181,A -85,B 0,C 180,E1 -4186.068,E2 -4186.068} C_VEL
LIN {X 0,Y 530.513,Z 719.475,A -85,B 0,C 180,E1 -4187.133,E2 -4187.133} C_VEL
LIN {X 0,Y 530.449,Z 723.659,A -85,B 0,C 180,E1 -4188.514,E2 -4188.514} C_VEL
LIN {X 0,Y 530.349,Z 725.777,A -85,B 0,C 180,E1 -4189.51,E2 -4189.51} C_VEL
LIN {X 0,Y 530.348,Z 727.157,A -85,B 0,C 180,E1 -4190.501,E2 -4190.501} C_VEL
LIN {X 0,Y 530.329,Z 727.886,A -85,B 0,C 180,E1 -4191.476,E2 -4191.476} C_VEL
LIN {X 0,Y 530.337,Z 727.867,A -85,B 0,C 180,E1 -4192.666,E2 -4192.666} C_VEL
LIN {X 0,Y 530.333,Z 726.764,A -85,B 0,C 180,E1 -4193.937,E2 -4193.937} C_VEL
LIN {X 0,Y 530.414,Z 724.38,A -85,B 0,C 180,E1 -4195.268,E2 -4195.268} C_VEL
LIN {X 0,Y 530.467,Z 720.754,A -85,B 0,C 180,E1 -4196.581,E2 -4196.581} C_VEL
LIN {X 0,Y 530.572,Z 715.255,A -85,B 0,C 180,E1 -4198.006,E2 -4198.006} C_VEL
LIN {X 0,Y 530.661,Z 709.246,A -85,B 0,C 180,E1 -4199.186,E2 -4199.186} C_VEL
LIN {X 0,Y 530.815,Z 701.115,A -85,B 0,C 180,E1 -4200.45,E2 -4200.45} C_VEL
LIN {X 0,Y 531.02,Z 692.315,A -85,B 0,C 180,E1 -4201.547,E2 -4201.547} C_VEL
LIN {X 0,Y 531.271,Z 682.967,A -85,B 0,C 180,E1 -4202.492,E2 -4202.492} C_VEL
LIN {X 0,Y 531.508,Z 672.11,A -85,B 0,C 180,E1 -4203.382,E2 -4203.382} C_VEL
LIN {X 0,Y 531.771,Z 661.481,A -85,B 0,C 180,E1 -4204.078,E2 -4204.078} C_VEL
LIN {X 0,Y 532.005,Z 649.642,A -85,B 0,C 180,E1 -4204.68,E2 -4204.68} C_VEL
LIN {X 0,Y 532.241,Z 636.759,A -85,B 0,C 180,E1 -4205.159,E2 -4205.159} C_VEL
LIN {X 0,Y 532.415,Z 624.04,A -85,B 0,C 180,E1 -4205.476,E2 -4205.476} C_VEL
LIN {X 0,Y 532.667,Z 526.794,A -85,B 0,C 180,E1 -4206.812,E2 -4206.812} C_VEL
LIN {X 0,Y 531.102,Z 518.459,A -85,B 0,C 180,E1 -4206.972,E2 -4206.972} C_VEL
LIN {X 0,Y 531.311,Z 506.571,A -85,B 0,C 180,E1 -4209.481,E2 -4209.481} C_VEL
LIN {X 0,Y 531.067,Z 503.336,A -85,B 0,C 180,E1 -4210.196,E2 -4210.196} C_VEL
LIN {X 0,Y 530.983,Z 503.346,A -85,B 0,C 180,E1 -4213.071,E2 -4213.071} C_VEL
LIN {X 0,Y 531.016,Z 503.335,A -85,B 0,C 180,E1 -4215.436,E2 -4215.436} C_VEL
LIN {X 0,Y 531.034,Z 503.336,A -85,B 0,C 180,E1 -4218.55,E2 -4218.55} C_VEL
LIN {X 0,Y 531.053,Z 503.33,A -85,B 0,C 180,E1 -4221.63,E2 -4221.63} C_VEL
LIN {X 0,Y 531.119,Z 503.327,A -85,B 0,C 180,E1 -4224.685,E2 -4224.685} C_VEL
LIN {X 0,Y 531.139,Z 503.319,A -85,B 0,C 180,E1 -4227.725,E2 -4227.725} C_VEL
LIN {X 0,Y 531.152,Z 503.324,A -85,B 0,C 180,E1 -4230.758,E2 -4230.758} C_VEL
LIN {X 0,Y 531.103,Z 503.331,A -85,B 0,C 180,E1 -4233.034,E2 -4233.034} C_VEL
LIN {X 0,Y 531.089,Z 503.325,A -85,B 0,C 180,E1 -4236.077,E2 -4236.077} C_VEL
LIN {X 0,Y 531.029,Z 503.339,A -85,B 0,C 180,E1 -4239.138,E2 -4239.138} C_VEL
LIN {X 0,Y 531.038,Z 503.332,A -85,B 0,C 180,E1 -4242.225,E2 -4242.225} C_VEL
LIN {X 0,Y 530.993,Z 503.34,A -85,B 0,C 180,E1 -4245.349,E2 -4245.349} C_VEL
LIN {X 0,Y 530.99,Z 503.34,A -85,B 0,C 180,E1 -4248.521,E2 -4248.521} C_VEL
LIN {X 0,Y 530.996,Z 503.345,A -85,B 0,C 180,E1 -4250.938,E2 -4250.938} C_VEL
LIN {X 0,Y 530.976,Z 503.339,A -85,B 0,C 180,E1 -4254.224,E2 -4254.224} C_VEL
LIN {X 0,Y 531.002,Z 503.341,A -85,B 0,C 180,E1 -4256.743,E2 -4256.743} C_VEL
LIN {X 0,Y 530.995,Z 503.341,A -85,B 0,C 180,E1 -4259.321,E2 -4259.321} C_VEL
LIN {X 0,Y 530.975,Z 503.339,A -85,B 0,C 180,E1 -4262.103,E2 -4262.103} C_VEL
LIN {X 0,Y 530.982,Z 503.345,A -85,B 0,C 180,E1 -4264.854,E2 -4264.854} C_VEL
LIN {X 0,Y 530.968,Z 503.342,A -85,B 0,C 180,E1 -4267.506,E2 -4267.506} C_VEL
LIN {X 0,Y 531.003,Z 503.337,A -85,B 0,C 180,E1 -4270.43,E2 -4270.43} C_VEL
LIN {X 0,Y 530.961,Z 503.344,A -85,B 0,C 180,E1 -4273.494,E2 -4273.494} C_VEL
LIN {X 0,Y 530.958,Z 503.343,A -85,B 0,C 180,E1 -4276.505,E2 -4276.505} C_VEL
LIN {X 0,Y 531,Z 503.338,A -85,B 0,C 180,E1 -4279.569,E2 -4279.569} C_VEL
LIN {X 0,Y 530.968,Z 503.342,A -85,B 0,C 180,E1 -4282.575,E2 -4282.575} C_VEL
LIN {X 0,Y 530.996,Z 503.342,A -85,B 0,C 180,E1 -4285.311,E2 -4285.311} C_VEL
LIN {X 0,Y 530.973,Z 503.339,A -85,B 0,C 180,E1 -4288.033,E2 -4288.033} C_VEL
LIN {X 0,Y 530.997,Z 503.342,A -85,B 0,C 180,E1 -4290.87,E2 -4290.87} C_VEL
LIN {X 0,Y 531.003,Z 503.343,A -85,B 0,C 180,E1 -4293.257,E2 -4293.257} C_VEL
LIN {X 0,Y 530.987,Z 503.337,A -85,B 0,C 180,E1 -4295.957,E2 -4295.957} C_VEL
LIN {X 0,Y 530.992,Z 503.345,A -85,B 0,C 180,E1 -4299.062,E2 -4299.062} C_VEL
LIN {X 0,Y 531.006,Z 503.335,A -85,B 0,C 180,E1 -4302.278,E2 -4302.278} C_VEL
LIN {X 0,Y 531.008,Z 503.34,A -85,B 0,C 180,E1 -4305.436,E2 -4305.436} C_VEL
LIN {X 0,Y 531.042,Z 503.332,A -85,B 0,C 180,E1 -4308.55,E2 -4308.55} C_VEL
LIN {X 0,Y 531.052,Z 503.332,A -85,B 0,C 180,E1 -4311.63,E2 -4311.63} C_VEL
LIN {X 0,Y 531.135,Z 503.321,A -85,B 0,C 180,E1 -4314.686,E2 -4314.686} C_VEL
LIN {X 0,Y 531.131,Z 503.322,A -85,B 0,C 180,E1 -4317.725,E2 -4317.725} C_VEL
LIN {X 0,Y 531.148,Z 503.32,A -85,B 0,C 180,E1 -4320.759,E2 -4320.759} C_VEL
LIN {X 0,Y 531.103,Z 503.329,A -85,B 0,C 180,E1 -4323.035,E2 -4323.035} C_VEL
LIN {X 0,Y 531.083,Z 503.325,A -85,B 0,C 180,E1 -4326.077,E2 -4326.077} C_VEL
LIN {X 0,Y 531.029,Z 503.34,A -85,B 0,C 180,E1 -4329.139,E2 -4329.139} C_VEL
LIN {X 0,Y 531.033,Z 503.332,A -85,B 0,C 180,E1 -4332.225,E2 -4332.225} C_VEL
LIN {X 0,Y 530.988,Z 503.345,A -85,B 0,C 180,E1 -4335.35,E2 -4335.35} C_VEL
LIN {X 0,Y 531.008,Z 503.338,A -85,B 0,C 180,E1 -4337.723,E2 -4337.723} C_VEL
LIN {X 0,Y 530.994,Z 503.341,A -85,B 0,C 180,E1 -4340.938,E2 -4340.938} C_VEL
LIN {X 0,Y 530.972,Z 503.339,A -85,B 0,C 180,E1 -4344.225,E2 -4344.225} C_VEL
LIN {X 0,Y 531.005,Z 503.337,A -85,B 0,C 180,E1 -4346.744,E2 -4346.744} C_VEL
LIN {X 0,Y 530.994,Z 503.346,A -85,B 0,C 180,E1 -4349.322,E2 -4349.322} C_VEL
LIN {X 0,Y 530.974,Z 503.339,A -85,B 0,C 180,E1 -4352.104,E2 -4352.104} C_VEL
LIN {X 0,Y 530.986,Z 503.34,A -85,B 0,C 180,E1 -4354.855,E2 -4354.855} C_VEL
LIN {X 0,Y 530.968,Z 503.346,A -85,B 0,C 180,E1 -4357.508,E2 -4357.508} C_VEL
LIN {X 0,Y 530.981,Z 503.338,A -85,B 0,C 180,E1 -4360.433,E2 -4360.433} C_VEL
LIN {X 0,Y 530.967,Z 503.349,A -85,B 0,C 180,E1 -4363.283,E2 -4363.283} C_VEL
LIN {X 0,Y 530.985,Z 503.343,A -85,B 0,C 180,E1 -4365.622,E2 -4365.622} C_VEL
LIN {X 0,Y 531.005,Z 503.335,A -85,B 0,C 180,E1 -4368.567,E2 -4368.567} C_VEL
LIN {X 0,Y 530.967,Z 503.349,A -85,B 0,C 180,E1 -4371.347,E2 -4371.347} C_VEL
LIN {X 0,Y 530.975,Z 503.339,A -85,B 0,C 180,E1 -4374.383,E2 -4374.383} C_VEL
LIN {X 0,Y 530.972,Z 503.346,A -85,B 0,C 180,E1 -4377.135,E2 -4377.135} C_VEL
LIN {X 0,Y 530.97,Z 503.345,A -85,B 0,C 180,E1 -4379.804,E2 -4379.804} C_VEL
LIN {X 0,Y 531.016,Z 503.337,A -85,B 0,C 180,E1 -4382.468,E2 -4382.468} C_VEL
LIN {X 0,Y 531.037,Z 503.406,A -85,B 0,C 180,E1 -4384.604,E2 -4384.604} C_VEL
LIN {X 0,Y 532.618,Z 511.24,A -85,B 0,C 180,E1 -4385.855,E2 -4385.855} C_VEL
LIN {X 0,Y 532.472,Z 523.161,A -85,B 0,C 180,E1 -4387.614,E2 -4387.614} C_VEL
LIN {X 0,Y 532.034,Z 541.87,A -85,B 0,C 180,E1 -4390.316,E2 -4390.316} C_VEL
LIN {X 0,Y 531.641,Z 562.721,A -85,B 0,C 180,E1 -4393.291,E2 -4393.291} C_VEL
LIN {X 0,Y 531.423,Z 575.125,A -85,B 0,C 180,E1 -4395.045,E2 -4395.045} C_VEL
LIN {X 0,Y 532.842,Z 585.139,A -85,B 0,C 180,E1 -4395.223,E2 -4395.223} C_VEL
LIN {X 0,Y 532.397,Z 683.873,A -85,B 0,C 180,E1 -4396.571,E2 -4396.571} C_VEL
LIN {X 0,Y 532.249,Z 697.191,A -85,B 0,C 180,E1 -4396.907,E2 -4396.907} C_VEL
LIN {X 0,Y 532.013,Z 709.375,A -85,B 0,C 180,E1 -4397.362,E2 -4397.362} C_VEL
LIN {X 0,Y 531.82,Z 720.766,A -85,B 0,C 180,E1 -4397.936,E2 -4397.936} C_VEL
LIN {X 0,Y 531.576,Z 731.905,A -85,B 0,C 180,E1 -4398.658,E2 -4398.658} C_VEL
LIN {X 0,Y 531.27,Z 742.538,A -85,B 0,C 180,E1 -4399.52,E2 -4399.52} C_VEL
LIN {X 0,Y 531.06,Z 752.115,A -85,B 0,C 180,E1 -4400.478,E2 -4400.478} C_VEL
LIN {X 0,Y 530.887,Z 759.962,A -85,B 0,C 180,E1 -4401.435,E2 -4401.435} C_VEL
LIN {X 0,Y 530.685,Z 767.622,A -85,B 0,C 180,E1 -4402.581,E2 -4402.581} C_VEL
LIN {X 0,Y 530.604,Z 774.68,A -85,B 0,C 180,E1 -4403.918,E2 -4403.918} C_VEL
LIN {X 0,Y 530.459,Z 779.373,A -85,B 0,C 180,E1 -4405.06,E2 -4405.06} C_VEL
LIN {X 0,Y 530.516,Z 782.958,A -85,B 0,C 180,E1 -4406.202,E2 -4406.202} C_VEL
LIN {X 0,Y 530.457,Z 784.807,A -85,B 0,C 180,E1 -4406.962,E2 -4406.962} C_VEL
LIN {X 0,Y 530.41,Z 786.194,A -85,B 0,C 180,E1 -4407.722,E2 -4407.722} C_VEL
LIN {X 0,Y 530.344,Z 787.786,A -85,B 0,C 180,E1 -4409.241,E2 -4409.241} C_VEL
LIN {X 0,Y 530.342,Z 788,A -85,B 0,C 180,E1 -4410,E2 -4410} C_VEL
LIN {X 0,Y 530.361,Z 787.184,A -85,B 0,C 180,E1 -4411.519,E2 -4411.519} C_VEL
LIN {X 0,Y 530.41,Z 786.196,A -85,B 0,C 180,E1 -4412.278,E2 -4412.278} C_VEL
LIN {X 0,Y 530.457,Z 784.81,A -85,B 0,C 180,E1 -4413.038,E2 -4413.038} C_VEL
LIN {X 0,Y 530.522,Z 781.896,A -85,B 0,C 180,E1 -4414.178,E2 -4414.178} C_VEL
LIN {X 0,Y 530.525,Z 777.948,A -85,B 0,C 180,E1 -4415.321,E2 -4415.321} C_VEL
LIN {X 0,Y 530.599,Z 772.265,A -85,B 0,C 180,E1 -4416.582,E2 -4416.582} C_VEL
LIN {X 0,Y 530.758,Z 765.236,A -85,B 0,C 180,E1 -4417.8,E2 -4417.8} C_VEL
LIN {X 0,Y 530.93,Z 756.994,A -85,B 0,C 180,E1 -4418.948,E2 -4418.948} C_VEL
LIN {X 0,Y 531.137,Z 748.542,A -85,B 0,C 180,E1 -4419.905,E2 -4419.905} C_VEL
LIN {X 0,Y 531.41,Z 738.094,A -85,B 0,C 180,E1 -4420.863,E2 -4420.863} C_VEL
LIN {X 0,Y 531.681,Z 727.139,A -85,B 0,C 180,E1 -4421.671,E2 -4421.671} C_VEL
LIN {X 0,Y 531.933,Z 716.409,A -85,B 0,C 180,E1 -4422.301,E2 -4422.301} C_VEL
LIN {X 0,Y 532.112,Z 704.765,A -85,B 0,C 180,E1 -4422.829,E2 -4422.829} C_VEL
LIN {X 0,Y 532.312,Z 691.29,A -85,B 0,C 180,E1 -4423.261,E2 -4423.261} C_VEL
LIN {X 0,Y 532.501,Z 677.984,A -85,B 0,C 180,E1 -4423.524,E2 -4423.524} C_VEL
LIN {X 0,Y 532.71,Z 583.351,A -85,B 0,C 180,E1 -4424.804,E2 -4424.804} C_VEL
LIN {X 0,Y 531.449,Z 574.979,A -85,B 0,C 180,E1 -4424.969,E2 -4424.969} C_VEL
LIN {X 0,Y 531.825,Z 552.554,A -85,B 0,C 180,E1 -4428.141,E2 -4428.141} C_VEL
LIN {X 0,Y 532.238,Z 531.939,A -85,B 0,C 180,E1 -4431.089,E2 -4431.089} C_VEL
LIN {X 0,Y 532.652,Z 513.744,A -85,B 0,C 180,E1 -4433.729,E2 -4433.729} C_VEL
LIN {X 0,Y 532.305,Z 509.633,A -85,B 0,C 180,E1 -4434.355,E2 -4434.355} C_VEL
LIN {X 0,Y 531.054,Z 503.336,A -85,B 0,C 180,E1 -4435.369,E2 -4435.369} C_VEL
LIN {X 0,Y 530.999,Z 503.345,A -85,B 0,C 180,E1 -4438.455,E2 -4438.455} C_VEL
LIN {X 0,Y 530.964,Z 503.346,A -85,B 0,C 180,E1 -4441.078,E2 -4441.078} C_VEL
LIN {X 0,Y 530.99,Z 503.34,A -85,B 0,C 180,E1 -4443.772,E2 -4443.772} C_VEL
LIN {X 0,Y 530.968,Z 503.349,A -85,B 0,C 180,E1 -4446.556,E2 -4446.556} C_VEL
LIN {X 0,Y 531.004,Z 503.336,A -85,B 0,C 180,E1 -4449.856,E2 -4449.856} C_VEL
LIN {X 0,Y 530.981,Z 503.345,A -85,B 0,C 180,E1 -4452.455,E2 -4452.455} C_VEL
LIN {X 0,Y 530.984,Z 503.338,A -85,B 0,C 180,E1 -4455.62,E2 -4455.62} C_VEL
LIN {X 0,Y 530.996,Z 503.342,A -85,B 0,C 180,E1 -4458.564,E2 -4458.564} C_VEL
LIN {X 0,Y 530.955,Z 503.342,A -85,B 0,C 180,E1 -4461.529,E2 -4461.529} C_VEL
LIN {X 0,Y 530.978,Z 503.342,A -85,B 0,C 180,E1 -4464.381,E2 -4464.381} C_VEL
LIN {X 0,Y 530.969,Z 503.345,A -85,B 0,C 180,E1 -4467.133,E2 -4467.133} C_VEL
LIN {X 0,Y 530.98,Z 503.338,A -85,B 0,C 180,E1 -4469.803,E2 -4469.803} C_VEL
LIN {X 0,Y 531.011,Z 503.338,A -85,B 0,C 180,E1 -4472.465,E2 -4472.465} C_VEL
LIN {X 0,Y 531.001,Z 503.342,A -85,B 0,C 180,E1 -4474.942,E2 -4474.942} C_VEL
LIN {X 0,Y 530.964,Z 503.342,A -85,B 0,C 180,E1 -4478.246,E2 -4478.246} C_VEL
LIN {X 0,Y 530.992,Z 503.342,A -85,B 0,C 180,E1 -4480.677,E2 -4480.677} C_VEL
LIN {X 0,Y 530.985,Z 503.345,A -85,B 0,C 180,E1 -4483.071,E2 -4483.071} C_VEL
LIN {X 0,Y 531.01,Z 503.336,A -85,B 0,C 180,E1 -4485.435,E2 -4485.435} C_VEL
LIN {X 0,Y 531.038,Z 503.335,A -85,B 0,C 180,E1 -4488.549,E2 -4488.549} C_VEL
LIN {X 0,Y 531.052,Z 503.331,A -85,B 0,C 180,E1 -4491.629,E2 -4491.629} C_VEL
LIN {X 0,Y 531.135,Z 503.323,A -85,B 0,C 180,E1 -4494.685,E2 -4494.685} C_VEL
LIN {X 0,Y 531.13,Z 503.32,A -85,B 0,C 180,E1 -4497.725,E2 -4497.725} C_VEL
LIN {X 0,Y 531.147,Z 503.323,A -85,B 0,C 180,E1 -4500.758,E2 -4500.758} C_VEL
LIN {X 0,Y 531.102,Z 503.331,A -85,B 0,C 180,E1 -4503.034,E2 -4503.034} C_VEL
LIN {X 0,Y 531.083,Z 503.325,A -85,B 0,C 180,E1 -4506.077,E2 -4506.077} C_VEL
LIN {X 0,Y 531.028,Z 503.341,A -85,B 0,C 180,E1 -4509.138,E2 -4509.138} C_VEL
LIN {X 0,Y 531.031,Z 503.333,A -85,B 0,C 180,E1 -4512.225,E2 -4512.225} C_VEL
LIN {X 0,Y 530.986,Z 503.344,A -85,B 0,C 180,E1 -4515.35,E2 -4515.35} C_VEL
LIN {X 0,Y 531.006,Z 503.338,A -85,B 0,C 180,E1 -4517.722,E2 -4517.722} C_VEL
LIN {X 0,Y 531.014,Z 503.335,A -85,B 0,C 180,E1 -4520.127,E2 -4520.127} C_VEL
LIN {X 0,Y 530.956,Z 503.35,A -85,B 0,C 180,E1 -4523.396,E2 -4523.396} C_VEL
LIN {X 0,Y 531.005,Z 503.339,A -85,B 0,C 180,E1 -4525.897,E2 -4525.897} C_VEL
LIN {X 0,Y 530.99,Z 503.341,A -85,B 0,C 180,E1 -4528.455,E2 -4528.455} C_VEL
LIN {X 0,Y 530.958,Z 503.35,A -85,B 0,C 180,E1 -4531.079,E2 -4531.079} C_VEL
LIN {X 0,Y 531.019,Z 503.455,A -85,B 0,C 180,E1 -4533.884,E2 -4533.884} C_VEL
LIN {X 0,Y 531.324,Z 507.071,A -85,B 0,C 180,E1 -4534.664,E2 -4534.664} C_VEL
LIN {X 0,Y 531.122,Z 518.46,A -85,B 0,C 180,E1 -4537.107,E2 -4537.107} C_VEL
LIN {X 0,Y 532.824,Z 528.162,A -85,B 0,C 180,E1 -4537.3,E2 -4537.3} C_VEL
LIN {X 0,Y 532.642,Z 574.205,A -85,B 0,C 180,E1 -4537.923,E2 -4537.923} C_VEL
LIN {X 0,Y 531.951,Z 580.051,A -85,B 0,C 180,E1 -4537.984,E2 -4537.984} C_VEL
LIN {X 0,Y 526.283,Z 599.048,A -85,B 0,C 180,E1 -4538.088,E2 -4538.088} C_VEL
LIN {X 0,Y 525.614,Z 604.892,A -85,B 0,C 180,E1 -4538.152,E2 -4538.152} C_VEL
LIN {X 0,Y 525.492,Z 626.656,A -85,B 0,C 180,E1 -4538.485,E2 -4538.485} C_VEL
LIN {X 0,Y 525.298,Z 639.698,A -85,B 0,C 180,E1 -4538.839,E2 -4538.839} C_VEL
LIN {X 0,Y 525.106,Z 651.677,A -85,B 0,C 180,E1 -4539.317,E2 -4539.317} C_VEL
LIN {X 0,Y 524.805,Z 663.313,A -85,B 0,C 180,E1 -4539.94,E2 -4539.94} C_VEL
LIN {X 0,Y 524.535,Z 674.524,A -85,B 0,C 180,E1 -4540.71,E2 -4540.71} C_VEL
LIN {X 0,Y 524.193,Z 684.859,A -85,B 0,C 180,E1 -4541.594,E2 -4541.594} C_VEL
LIN {X 0,Y 523.988,Z 694.217,A -85,B 0,C 180,E1 -4542.593,E2 -4542.593} C_VEL
LIN {X 0,Y 523.724,Z 703.042,A -85,B 0,C 180,E1 -4543.756,E2 -4543.756} C_VEL
LIN {X 0,Y 523.61,Z 709.73,A -85,B 0,C 180,E1 -4544.847,E2 -4544.847} C_VEL
LIN {X 0,Y 523.499,Z 715.98,A -85,B 0,C 180,E1 -4546.127,E2 -4546.127} C_VEL
LIN {X 0,Y 523.423,Z 720.182,A -85,B 0,C 180,E1 -4547.225,E2 -4547.225} C_VEL
LIN {X 0,Y 523.367,Z 723.431,A -85,B 0,C 180,E1 -4548.327,E2 -4548.327} C_VEL
LIN {X 0,Y 523.234,Z 726.597,A -85,B 0,C 180,E1 -4549.961,E2 -4549.961} C_VEL
LIN {X 0,Y 523.214,Z 727.781,A -85,B 0,C 180,E1 -4551.175,E2 -4551.175} C_VEL
LIN {X 0,Y 523.229,Z 727.983,A -85,B 0,C 180,E1 -4552.418,E2 -4552.418} C_VEL
LIN {X 0,Y 523.236,Z 727.051,A -85,B 0,C 180,E1 -4553.773,E2 -4553.773} C_VEL
LIN {X 0,Y 523.278,Z 725.113,A -85,B 0,C 180,E1 -4555.011,E2 -4555.011} C_VEL
LIN {X 0,Y 523.391,Z 721.787,A -85,B 0,C 180,E1 -4556.358,E2 -4556.358} C_VEL
LIN {X 0,Y 523.463,Z 716.807,A -85,B 0,C 180,E1 -4557.761,E2 -4557.761} C_VEL
LIN {X 0,Y 523.565,Z 711.776,A -85,B 0,C 180,E1 -4558.852,E2 -4558.852} C_VEL
LIN {X 0,Y 523.735,Z 705.14,A -85,B 0,C 180,E1 -4560.01,E2 -4560.01} C_VEL
LIN {X 0,Y 523.903,Z 697.259,A -85,B 0,C 180,E1 -4561.124,E2 -4561.124} C_VEL
LIN {X 0,Y 524.19,Z 687.411,A -85,B 0,C 180,E1 -4562.236,E2 -4562.236} C_VEL
LIN {X 0,Y 524.481,Z 676.538,A -85,B 0,C 180,E1 -4563.22,E2 -4563.22} C_VEL
LIN {X 0,Y 524.744,Z 665.94,A -85,B 0,C 180,E1 -4563.984,E2 -4563.984} C_VEL
LIN {X 0,Y 525.016,Z 654.413,A -85,B 0,C 180,E1 -4564.637,E2 -4564.637} C_VEL
LIN {X 0,Y 525.248,Z 642.996,A -85,B 0,C 180,E1 -4565.131,E2 -4565.131} C_VEL
LIN {X 0,Y 525.422,Z 630.395,A -85,B 0,C 180,E1 -4565.521,E2 -4565.521} C_VEL
LIN {X 0,Y 525.594,Z 616.597,A -85,B 0,C 180,E1 -4565.775,E2 -4565.775} C_VEL
LIN {X 0,Y 525.905,Z 528.132,A -85,B 0,C 180,E1 -4566.991,E2 -4566.991} C_VEL
LIN {X 0,Y 524.127,Z 518.627,A -85,B 0,C 180,E1 -4567.2,E2 -4567.2} C_VEL
LIN {X 0,Y 524.293,Z 506.63,A -85,B 0,C 180,E1 -4569.772,E2 -4569.772} C_VEL
LIN {X 0,Y 524.011,Z 504.215,A -85,B 0,C 180,E1 -4570.334,E2 -4570.334} C_VEL
LIN {X 0,Y 523.964,Z 504.221,A -85,B 0,C 180,E1 -4572.838,E2 -4572.838} C_VEL
LIN {X 0,Y 523.974,Z 504.215,A -85,B 0,C 180,E1 -4575.236,E2 -4575.236} C_VEL
LIN {X 0,Y 524.009,Z 504.209,A -85,B 0,C 180,E1 -4578.394,E2 -4578.394} C_VEL
LIN {X 0,Y 524.001,Z 504.209,A -85,B 0,C 180,E1 -4581.516,E2 -4581.516} C_VEL
LIN {X 0,Y 524.08,Z 504.203,A -85,B 0,C 180,E1 -4584.614,E2 -4584.614} C_VEL
LIN {X 0,Y 524.111,Z 504.194,A -85,B 0,C 180,E1 -4587.695,E2 -4587.695} C_VEL
LIN {X 0,Y 524.122,Z 504.2,A -85,B 0,C 180,E1 -4590.768,E2 -4590.768} C_VEL
LIN {X 0,Y 524.07,Z 504.206,A -85,B 0,C 180,E1 -4593.075,E2 -4593.075} C_VEL
LIN {X 0,Y 524.05,Z 504.202,A -85,B 0,C 180,E1 -4596.159,E2 -4596.159} C_VEL
LIN {X 0,Y 523.997,Z 504.213,A -85,B 0,C 180,E1 -4599.262,E2 -4599.262} C_VEL
LIN {X 0,Y 524,Z 504.208,A -85,B 0,C 180,E1 -4601.739,E2 -4601.739} C_VEL
LIN {X 0,Y 523.99,Z 504.217,A -85,B 0,C 180,E1 -4605.052,E2 -4605.052} C_VEL
LIN {X 0,Y 523.961,Z 504.212,A -85,B 0,C 180,E1 -4607.969,E2 -4607.969} C_VEL
LIN {X 0,Y 523.968,Z 504.213,A -85,B 0,C 180,E1 -4610.41,E2 -4610.41} C_VEL
LIN {X 0,Y 523.913,Z 504.227,A -85,B 0,C 180,E1 -4612.893,E2 -4612.893} C_VEL
LIN {X 0,Y 523.948,Z 504.217,A -85,B 0,C 180,E1 -4615.418,E2 -4615.418} C_VEL
LIN {X 0,Y 523.965,Z 504.212,A -85,B 0,C 180,E1 -4617.998,E2 -4617.998} C_VEL
LIN {X 0,Y 523.947,Z 504.221,A -85,B 0,C 180,E1 -4620.856,E2 -4620.856} C_VEL
LIN {X 0,Y 523.955,Z 504.214,A -85,B 0,C 180,E1 -4623.734,E2 -4623.734} C_VEL
LIN {X 0,Y 523.919,Z 504.219,A -85,B 0,C 180,E1 -4626.404,E2 -4626.404} C_VEL
LIN {X 0,Y 523.953,Z 504.223,A -85,B 0,C 180,E1 -4629.081,E2 -4629.081} C_VEL
LIN {X 0,Y 523.959,Z 504.213,A -85,B 0,C 180,E1 -4632.117,E2 -4632.117} C_VEL
LIN {X 0,Y 523.948,Z 504.22,A -85,B 0,C 180,E1 -4635.308,E2 -4635.308} C_VEL
LIN {X 0,Y 523.964,Z 504.216,A -85,B 0,C 180,E1 -4638.687,E2 -4638.687} C_VEL
LIN {X 0,Y 523.945,Z 504.224,A -85,B 0,C 180,E1 -4641.075,E2 -4641.075} C_VEL
LIN {X 0,Y 523.921,Z 504.218,A -85,B 0,C 180,E1 -4643.828,E2 -4643.828} C_VEL
LIN {X 0,Y 523.935,Z 504.219,A -85,B 0,C 180,E1 -4646.636,E2 -4646.636} C_VEL
LIN {X 0,Y 523.954,Z 504.219,A -85,B 0,C 180,E1 -4649.356,E2 -4649.356} C_VEL
LIN {X 0,Y 523.97,Z 504.212,A -85,B 0,C 180,E1 -4652.28,E2 -4652.28} C_VEL
LIN {X 0,Y 523.948,Z 504.216,A -85,B 0,C 180,E1 -4654.582,E2 -4654.582} C_VEL
LIN {X 0,Y 523.907,Z 504.229,A -85,B 0,C 180,E1 -4657.107,E2 -4657.107} C_VEL
LIN {X 0,Y 523.969,Z 504.212,A -85,B 0,C 180,E1 -4659.866,E2 -4659.866} C_VEL
LIN {X 0,Y 523.961,Z 504.217,A -85,B 0,C 180,E1 -4662.837,E2 -4662.837} C_VEL
LIN {X 0,Y 523.966,Z 504.22,A -85,B 0,C 180,E1 -4665.236,E2 -4665.236} C_VEL
LIN {X 0,Y 524.002,Z 504.208,A -85,B 0,C 180,E1 -4668.394,E2 -4668.394} C_VEL
LIN {X 0,Y 523.999,Z 504.212,A -85,B 0,C 180,E1 -4671.516,E2 -4671.516} C_VEL
LIN {X 0,Y 524.094,Z 504.198,A -85,B 0,C 180,E1 -4674.614,E2 -4674.614} C_VEL
LIN {X 0,Y 524.103,Z 504.197,A -85,B 0,C 180,E1 -4677.695,E2 -4677.695} C_VEL
LIN {X 0,Y 524.117,Z 504.196,A -85,B 0,C 180,E1 -4680.769,E2 -4680.769} C_VEL
LIN {X 0,Y 524.07,Z 504.206,A -85,B 0,C 180,E1 -4683.075,E2 -4683.075} C_VEL
LIN {X 0,Y 524.044,Z 504.202,A -85,B 0,C 180,E1 -4686.159,E2 -4686.159} C_VEL
LIN {X 0,Y 523.997,Z 504.217,A -85,B 0,C 180,E1 -4689.262,E2 -4689.262} C_VEL
LIN {X 0,Y 523.999,Z 504.21,A -85,B 0,C 180,E1 -4691.743,E2 -4691.743} C_VEL
LIN {X 0,Y 523.983,Z 504.216,A -85,B 0,C 180,E1 -4695.053,E2 -4695.053} C_VEL
LIN {X 0,Y 523.956,Z 504.214,A -85,B 0,C 180,E1 -4697.97,E2 -4697.97} C_VEL
LIN {X 0,Y 523.965,Z 504.212,A -85,B 0,C 180,E1 -4700.411,E2 -4700.411} C_VEL
LIN {X 0,Y 523.909,Z 504.223,A -85,B 0,C 180,E1 -4702.894,E2 -4702.894} C_VEL
LIN {X 0,Y 523.948,Z 504.222,A -85,B 0,C 180,E1 -4705.419,E2 -4705.419} C_VEL
LIN {X 0,Y 523.964,Z 504.213,A -85,B 0,C 180,E1 -4708,E2 -4708} C_VEL
LIN {X 0,Y 523.946,Z 504.217,A -85,B 0,C 180,E1 -4710.857,E2 -4710.857} C_VEL
LIN {X 0,Y 523.957,Z 504.216,A -85,B 0,C 180,E1 -4713.736,E2 -4713.736} C_VEL
LIN {X 0,Y 523.918,Z 504.218,A -85,B 0,C 180,E1 -4716.405,E2 -4716.405} C_VEL
LIN {X 0,Y 523.919,Z 504.223,A -85,B 0,C 180,E1 -4719.085,E2 -4719.085} C_VEL
LIN {X 0,Y 523.953,Z 504.214,A -85,B 0,C 180,E1 -4722.119,E2 -4722.119} C_VEL
LIN {X 0,Y 523.953,Z 504.223,A -85,B 0,C 180,E1 -4725.31,E2 -4725.31} C_VEL
LIN {X 0,Y 523.97,Z 504.212,A -85,B 0,C 180,E1 -4728.688,E2 -4728.688} C_VEL
LIN {X 0,Y 523.924,Z 504.222,A -85,B 0,C 180,E1 -4731.08,E2 -4731.08} C_VEL
LIN {X 0,Y 523.923,Z 504.22,A -85,B 0,C 180,E1 -4733.828,E2 -4733.828} C_VEL
LIN {X 0,Y 523.942,Z 504.217,A -85,B 0,C 180,E1 -4736.637,E2 -4736.637} C_VEL
LIN {X 0,Y 523.957,Z 504.222,A -85,B 0,C 180,E1 -4739.357,E2 -4739.357} C_VEL
LIN {X 0,Y 523.979,Z 504.214,A -85,B 0,C 180,E1 -4742.282,E2 -4742.282} C_VEL
LIN {X 0,Y 524.011,Z 504.342,A -85,B 0,C 180,E1 -4744.429,E2 -4744.429} C_VEL
LIN {X 0,Y 525.746,Z 513.717,A -85,B 0,C 180,E1 -4745.939,E2 -4745.939} C_VEL
LIN {X 0,Y 525.444,Z 527.589,A -85,B 0,C 180,E1 -4748.007,E2 -4748.007} C_VEL
LIN {X 0,Y 524.981,Z 547.098,A -85,B 0,C 180,E1 -4750.854,E2 -4750.854} C_VEL
LIN {X 0,Y 524.507,Z 569.321,A -85,B 0,C 180,E1 -4754.057,E2 -4754.057} C_VEL
LIN {X 0,Y 524.416,Z 575.006,A -85,B 0,C 180,E1 -4754.848,E2 -4754.848} C_VEL
LIN {X 0,Y 525.971,Z 585.386,A -85,B 0,C 180,E1 -4755.036,E2 -4755.036} C_VEL
LIN {X 0,Y 525.473,Z 683.316,A -85,B 0,C 180,E1 -4756.39,E2 -4756.39} C_VEL
LIN {X 0,Y 525.323,Z 696.689,A -85,B 0,C 180,E1 -4756.731,E2 -4756.731} C_VEL
LIN {X 0,Y 525.029,Z 710.044,A -85,B 0,C 180,E1 -4757.24,E2 -4757.24} C_VEL
LIN {X 0,Y 524.819,Z 721.536,A -85,B 0,C 180,E1 -4757.841,E2 -4757.841} C_VEL
LIN {X 0,Y 524.523,Z 732.913,A -85,B 0,C 180,E1 -4758.602,E2 -4758.602} C_VEL
LIN {X 0,Y 524.224,Z 743.407,A -85,B 0,C 180,E1 -4759.475,E2 -4759.475} C_VEL
LIN {X 0,Y 524.026,Z 751.994,A -85,B 0,C 180,E1 -4760.349,E2 -4760.349} C_VEL
LIN {X 0,Y 523.852,Z 759.918,A -85,B 0,C 180,E1 -4761.319,E2 -4761.319} C_VEL
LIN {X 0,Y 523.633,Z 767.622,A -85,B 0,C 180,E1 -4762.481,E2 -4762.481} C_VEL
LIN {X 0,Y 523.515,Z 774.68,A -85,B 0,C 180,E1 -4763.835,E2 -4763.835} C_VEL
LIN {X 0,Y 523.384,Z 779.373,A -85,B 0,C 180,E1 -4764.993,E2 -4764.993} C_VEL
LIN {X 0,Y 523.443,Z 782.958,A -85,B 0,C 180,E1 -4766.151,E2 -4766.151} C_VEL
LIN {X 0,Y 523.368,Z 784.807,A -85,B 0,C 180,E1 -4766.921,E2 -4766.921} C_VEL
LIN {X 0,Y 523.334,Z 786.193,A -85,B 0,C 180,E1 -4767.691,E2 -4767.691} C_VEL
LIN {X 0,Y 523.25,Z 787.785,A -85,B 0,C 180,E1 -4769.23,E2 -4769.23} C_VEL
LIN {X 0,Y 523.246,Z 788,A -85,B 0,C 180,E1 -4770,E2 -4770} C_VEL
LIN {X 0,Y 523.274,Z 787.183,A -85,B 0,C 180,E1 -4771.539,E2 -4771.539} C_VEL
LIN {X 0,Y 523.334,Z 786.196,A -85,B 0,C 180,E1 -4772.309,E2 -4772.309} C_VEL
LIN {X 0,Y 523.368,Z 784.81,A -85,B 0,C 180,E1 -4773.079,E2 -4773.079} C_VEL
LIN {X 0,Y 523.441,Z 781.895,A -85,B 0,C 180,E1 -4774.235,E2 -4774.235} C_VEL
LIN {X 0,Y 523.464,Z 777.948,A -85,B 0,C 180,E1 -4775.393,E2 -4775.393} C_VEL
LIN {X 0,Y 523.523,Z 772.729,A -85,B 0,C 180,E1 -4776.58,E2 -4776.58} C_VEL
LIN {X 0,Y 523.665,Z 766.466,A -85,B 0,C 180,E1 -4777.713,E2 -4777.713} C_VEL
LIN {X 0,Y 523.852,Z 758.417,A -85,B 0,C 180,E1 -4778.875,E2 -4778.875} C_VEL
LIN {X 0,Y 524.078,Z 750.191,A -85,B 0,C 180,E1 -4779.845,E2 -4779.845} C_VEL
LIN {X 0,Y 524.334,Z 740.16,A -85,B 0,C 180,E1 -4780.815,E2 -4780.815} C_VEL
LIN {X 0,Y 524.631,Z 728.746,A -85,B 0,C 180,E1 -4781.696,E2 -4781.696} C_VEL
LIN {X 0,Y 524.892,Z 717.746,A -85,B 0,C 180,E1 -4782.37,E2 -4782.37} C_VEL
LIN {X 0,Y 525.138,Z 705.457,A -85,B 0,C 180,E1 -4782.954,E2 -4782.954} C_VEL
LIN {X 0,Y 525.346,Z 692.541,A -85,B 0,C 180,E1 -4783.391,E2 -4783.391} C_VEL
LIN {X 0,Y 525.581,Z 678.832,A -85,B 0,C 180,E1 -4783.681,E2 -4783.681} C_VEL
LIN {X 0,Y 525.851,Z 584.158,A -85,B 0,C 180,E1 -4784.982,E2 -4784.982} C_VEL
LIN {X 0,Y 524.388,Z 574.576,A -85,B 0,C 180,E1 -4785.17,E2 -4785.17} C_VEL
LIN {X 0,Y 524.821,Z 552.774,A -85,B 0,C 180,E1 -4788.301,E2 -4788.301} C_VEL
LIN {X 0,Y 525.267,Z 532.934,A -85,B 0,C 180,E1 -4791.177,E2 -4791.177} C_VEL
LIN {X 0,Y 525.71,Z 514.773,A -85,B 0,C 180,E1 -4793.853,E2 -4793.853} C_VEL
LIN {X 0,Y 525.239,Z 510.541,A -85,B 0,C 180,E1 -4794.511,E2 -4794.511} C_VEL
LIN {X 0,Y 524.011,Z 504.213,A -85,B 0,C 180,E1 -4795.549,E2 -4795.549} C_VEL
LIN {X 0,Y 523.97,Z 504.216,A -85,B 0,C 180,E1 -4797.998,E2 -4797.998} C_VEL
LIN {X 0,Y 523.947,Z 504.223,A -85,B 0,C 180,E1 -4800.854,E2 -4800.854} C_VEL
LIN {X 0,Y 523.961,Z 504.216,A -85,B 0,C 180,E1 -4803.734,E2 -4803.734} C_VEL
LIN {X 0,Y 523.922,Z 504.225,A -85,B 0,C 180,E1 -4806.403,E2 -4806.403} C_VEL
LIN {X 0,Y 523.93,Z 504.221,A -85,B 0,C 180,E1 -4809.083,E2 -4809.083} C_VEL
LIN {X 0,Y 523.97,Z 504.214,A -85,B 0,C 180,E1 -4811.312,E2 -4811.312} C_VEL
LIN {X 0,Y 523.953,Z 504.223,A -85,B 0,C 180,E1 -4814.69,E2 -4814.69} C_VEL
LIN {X 0,Y 523.953,Z 504.213,A -85,B 0,C 180,E1 -4817.881,E2 -4817.881} C_VEL
LIN {X 0,Y 523.92,Z 504.226,A -85,B 0,C 180,E1 -4820.915,E2 -4820.915} C_VEL
LIN {X 0,Y 523.923,Z 504.217,A -85,B 0,C 180,E1 -4823.827,E2 -4823.827} C_VEL
LIN {X 0,Y 523.938,Z 504.221,A -85,B 0,C 180,E1 -4826.635,E2 -4826.635} C_VEL
LIN {X 0,Y 523.958,Z 504.215,A -85,B 0,C 180,E1 -4829.355,E2 -4829.355} C_VEL
LIN {X 0,Y 523.974,Z 504.213,A -85,B 0,C 180,E1 -4832.28,E2 -4832.28} C_VEL
LIN {X 0,Y 523.948,Z 504.22,A -85,B 0,C 180,E1 -4834.581,E2 -4834.581} C_VEL
LIN {X 0,Y 523.909,Z 504.225,A -85,B 0,C 180,E1 -4837.106,E2 -4837.106} C_VEL
LIN {X 0,Y 523.971,Z 504.211,A -85,B 0,C 180,E1 -4839.865,E2 -4839.865} C_VEL
LIN {X 0,Y 523.963,Z 504.22,A -85,B 0,C 180,E1 -4842.837,E2 -4842.837} C_VEL
LIN {X 0,Y 523.967,Z 504.216,A -85,B 0,C 180,E1 -4845.235,E2 -4845.235} C_VEL
LIN {X 0,Y 524.002,Z 504.21,A -85,B 0,C 180,E1 -4848.394,E2 -4848.394} C_VEL
LIN {X 0,Y 523.999,Z 504.21,A -85,B 0,C 180,E1 -4851.516,E2 -4851.516} C_VEL
LIN {X 0,Y 524.094,Z 504.199,A -85,B 0,C 180,E1 -4854.613,E2 -4854.613} C_VEL
LIN {X 0,Y 524.103,Z 504.196,A -85,B 0,C 180,E1 -4857.694,E2 -4857.694} C_VEL
LIN {X 0,Y 524.117,Z 504.198,A -85,B 0,C 180,E1 -4860.768,E2 -4860.768} C_VEL
LIN {X 0,Y 524.069,Z 504.207,A -85,B 0,C 180,E1 -4863.075,E2 -4863.075} C_VEL
LIN {X 0,Y 524.043,Z 504.202,A -85,B 0,C 180,E1 -4866.159,E2 -4866.159} C_VEL
LIN {X 0,Y 523.995,Z 504.216,A -85,B 0,C 180,E1 -4869.262,E2 -4869.262} C_VEL
LIN {X 0,Y 523.998,Z 504.21,A -85,B 0,C 180,E1 -4871.743,E2 -4871.743} C_VEL
LIN {X 0,Y 523.982,Z 504.22,A -85,B 0,C 180,E1 -4875.052,E2 -4875.052} C_VEL
LIN {X 0,Y 523.955,Z 504.215,A -85,B 0,C 180,E1 -4877.969,E2 -4877.969} C_VEL
LIN {X 0,Y 523.962,Z 504.214,A -85,B 0,C 180,E1 -4880.41,E2 -4880.41} C_VEL
LIN {X 0,Y 523.907,Z 504.227,A -85,B 0,C 180,E1 -4882.893,E2 -4882.893} C_VEL
